    report_progress()
    set_digital_out(0, True)
    new_pose = pose_trans(tuft_coords, p[0.5915, 0.8585, -0.0020, 0, 0, 0])
    movel(p[new_pose[0], new_pose[1], new_pose[2], current_pose[3], current_pose[4], current_pose[5]], a=1.2, v=0.0600)
    report_progress()
    set_digital_out(0, False)
    new_pose = pose_trans(tuft_coords, p[0.5915, 0.8585, 0.1500, 0, 0, 0])
    movel(p[new_pose[0], new_pose[1], new_pose[2], current_pose[3], current_pose[4], current_pose[5]], a=0.8, v=0.2000)
    report_progress()
    new_pose = pose_trans(tuft_coords, p[0.5935, 0.1895, 0.1500, 0, 0, 0])
    movel(p[new_pose[0], new_pose[1], new_pose[2], current_pose[3], current_pose[4], current_pose[5]], a=1.2, v=0.2000)
    report_progress()
    new_pose = pose_trans(tuft_coords, p[0.5935, 0.1895, -0.0020, 0, 0, 0])
    movel(p[new_pose[0], new_pose[1], new_pose[2], current_pose[3], current_pose[4], current_pose[5]], a=0.8, v=0.2000)
    report_progress()
    set_digital_out(0, True)
    new_pose = pose_trans(tuft_coords, p[0.5935, 0.8605, -0.0020, 0, 0, 0])
    movel(p[new_pose[0], new_pose[1], new_pose[2], current_pose[3], current_pose[4], current_pose[5]], a=1.2, v=0.0600)
    report_progress()
    set_digital_out(0, False)
    new_pose = pose_trans(tuft_coords, p[0.5935, 0.8605, 0.1500, 0, 0, 0])
    movel(p[new_pose[0], new_pose[1], new_pose[2], current_pose[3], current_pose[4], current_pose[5]], a=0.8, v=0.2000)
    report_progress()
    new_pose = pose_trans(tuft_coords, p[0.5954, 0.1895, 0.1500, 0, 0, 0])
    movel(p[new_pose[0], new_pose[1], new_pose[2], current_pose[3], current_pose[4], current_pose[5]], a=1.2, v=0.2000)
    report_progress()
    new_pose = pose_trans(tuft_coords, p[0.5954, 0.1895, -0.0020, 0, 0, 0])
    movel(p[new_pose[0], new_pose[1], new_pose[2], current_pose[3], current_pose[4], current_pose[5]], a=0.8, v=0.2000)
    report_progress()
    set_digital_out(0, True)
    new_pose = pose_trans(tuft_coords, p[0.5954, 0.8605, -0.0020, 0, 0, 0])
    movel(p[new_pose[0], new_pose[1], new_pose[2], current_pose[3], current_pose[4], current_pose[5]], a=1.2, v=0.0600)
    report_progress()
    set_digital_out(0, False)
    new_pose = pose_trans(tuft_coords, p[0.5954, 0.8605, 0.1500, 0, 0, 0])
    movel(p[new_pose[0], new_pose[1], new_pose[2], current_pose[3], current_pose[4], current_pose[5]], a=0.8, v=0.2000)
    report_progress()
    new_pose = pose_trans(tuft_coords, p[0.5974, 0.1876, 0.1500, 0, 0, 0])
    movel(p[new_pose[0], new_pose[1], new_pose[2], current_pose[3], current_pose[4], current_pose[5]], a=1.2, v=0.2000)
    report_progress()
    new_pose = pose_trans(tuft_coords, p[0.5974, 0.1876, -0.0020, 0, 0, 0])
    movel(p[new_pose[0], new_pose[1], new_pose[2], current_pose[3], current_pose[4], current_pose[5]], a=0.8, v=0.2000)
    report_progress()
    set_digital_out(0, True)
    new_pose = pose_trans(tuft_coords, p[0.5974, 0.8624, -0.0020, 0, 0, 0])
    movel(p[new_pose[0], new_pose[1], new_pose[2], current_pose[3], current_pose[4], current_pose[5]], a=1.2, v=0.0600)
    report_progress()
    set_digital_out(0, False)
    new_pose = pose_trans(tuft_coords, p[0.5974, 0.8624, 0.1500, 0, 0, 0])
    movel(p[new_pose[0], new_pose[1], new_pose[2], current_pose[3], current_pose[4], current_pose[5]], a=0.8, v=0.2000)
    report_progress()
    new_pose = pose_trans(tuft_coords, p[0.5993, 0.1876, 0.1500, 0, 0, 0])
    movel(p[new_pose[0], new_pose[1], new_pose[2], current_pose[3], current_pose[4], current_pose[5]], a=1.2, v=0.2000)
    report_progress()
    new_pose = pose_trans(tuft_coords, p[0.5993, 0.1876, -0.0020, 0, 0, 0])
    movel(p[new_pose[0], new_pose[1], new_pose[2], current_pose[3], current_pose[4], current_pose[5]], a=0.8, v=0.2000)
    report_progress()
    set_digital_out(0, True)
    new_pose = pose_trans(tuft_coords, p[0.5993, 0.8624, -0.0020, 0, 0, 0])
    movel(p[new_pose[0], new_pose[1], new_pose[2], current_pose[3], current_pose[4], current_pose[5]], a=1.2, v=0.0600)
    report_progress()
    set_digital_out(0, False)
    new_pose = pose_trans(tuft_coords, p[0.5993, 0.8624, 0.1500, 0, 0, 0])
    movel(p[new_pose[0], new_pose[1], new_pose[2], current_pose[3], current_pose[4], current_pose[5]], a=0.8, v=0.2000)
    report_progress()
    new_pose = pose_trans(tuft_coords, p[0.6012, 0.1856, 0.1500, 0, 0, 0])
    movel(p[new_pose[0], new_pose[1], new_pose[2], current_pose[3], current_pose[4], current_pose[5]], a=1.2, v=0.2000)
    report_progress()
    new_pose = pose_trans(tuft_coords, p[0.6012, 0.1856, -0.0020, 0, 0, 0])
    movel(p[new_pose[0], new_pose[1], new_pose[2], current_pose[3], current_pose[4], current_pose[5]], a=0.8, v=0.2000)
    report_progress()
    set_digital_out(0, True)
    new_pose = pose_trans(tuft_coords, p[0.6012, 0.8644, -0.0020, 0, 0, 0])
    movel(p[new_pose[0], new_pose[1], new_pose[2], current_pose[3], current_pose[4], current_pose[5]], a=1.2, v=0.0600)
    report_progress()
    set_digital_out(0, False)
    new_pose = pose_trans(tuft_coords, p[0.6012, 0.8644, 0.1500, 0, 0, 0])
    movel(p[new_pose[0], new_pose[1], new_pose[2], current_pose[3], current_pose[4], current_pose[5]], a=0.8, v=0.2000)
    report_progress()
    new_pose = pose_trans(tuft_coords, p[0.6032, 0.1856, 0.1500, 0, 0, 0])
    movel(p[new_pose[0], new_pose[1], new_pose[2], current_pose[3], current_pose[4], current_pose[5]], a=1.2, v=0.2000)
    report_progress()
    new_pose = pose_trans(tuft_coords, p[0.6032, 0.1856, -0.0020, 0, 0, 0])
    movel(p[new_pose[0], new_pose[1], new_pose[2], current_pose[3], current_pose[4], current_pose[5]], a=0.8, v=0.2000)
    report_progress()
    set_digital_out(0, True)
    new_pose = pose_trans(tuft_coords, p[0.6032, 0.8644, -0.0020, 0, 0, 0])
    movel(p[new_pose[0], new_pose[1], new_pose[2], current_pose[3], current_pose[4], current_pose[5]], a=1.2, v=0.0600)
    report_progress()
    set_digital_out(0, False)
    new_pose = pose_trans(tuft_coords, p[0.6032, 0.8644, 0.1500, 0, 0, 0])
    movel(p[new_pose[0], new_pose[1], new_pose[2], current_pose[3], current_pose[4], current_pose[5]], a=0.8, v=0.2000)
    report_progress()
    new_pose = pose_trans(tuft_coords, p[0.6051, 0.1856, 0.1500, 0, 0, 0])
    movel(p[new_pose[0], new_pose[1], new_pose[2], current_pose[3], current_pose[4], current_pose[5]], a=1.2, v=0.2000)
    report_progress()
    new_pose = pose_trans(tuft_coords, p[0.6051, 0.1856, -0.0020, 0, 0, 0])
    movel(p[new_pose[0], new_pose[1], new_pose[2], current_pose[3], current_pose[4], current_pose[5]], a=0.8, v=0.2000)
    report_progress()
    set_digital_out(0, True)
    new_pose = pose_trans(tuft_coords, p[0.6051, 0.8644, -0.0020, 0, 0, 0])
    movel(p[new_pose[0], new_pose[1], new_pose[2], current_pose[3], current_pose[4], current_pose[5]], a=1.2, v=0.0600)
    report_progress()
    set_digital_out(0, False)
    new_pose = pose_trans(tuft_coords, p[0.6051, 0.8644, 0.1500, 0, 0, 0])
    movel(p[new_pose[0], new_pose[1], new_pose[2], current_pose[3], current_pose[4], current_pose[5]], a=0.8, v=0.2000)
    report_progress()
    new_pose = pose_trans(tuft_coords, p[0.6071, 0.1836, 0.1500, 0, 0, 0])
    movel(p[new_pose[0], new_pose[1], new_pose[2], current_pose[3], current_pose[4], current_pose[5]], a=1.2, v=0.2000)
    report_progress()
    new_pose = pose_trans(tuft_coords, p[0.6071, 0.1836, -0.0020, 0, 0, 0])
    movel(p[new_pose[0], new_pose[1], new_pose[2], current_pose[3], current_pose[4], current_pose[5]], a=0.8, v=0.2000)
    report_progress()
    set_digital_out(0, True)
    new_pose = pose_trans(tuft_coords, p[0.6071, 0.8664, -0.0020, 0, 0, 0])
    movel(p[new_pose[0], new_pose[1], new_pose[2], current_pose[3], current_pose[4], current_pose[5]], a=1.2, v=0.0600)
    report_progress()
    set_digital_out(0, False)
    new_pose = pose_trans(tuft_coords, p[0.6071, 0.8664, 0.1500, 0, 0, 0])
    movel(p[new_pose[0], new_pose[1], new_pose[2], current_pose[3], current_pose[4], current_pose[5]], a=0.8, v=0.2000)
    report_progress()
    new_pose = pose_trans(tuft_coords, p[0.6090, 0.1836, 0.1500, 0, 0, 0])
    movel(p[new_pose[0], new_pose[1], new_pose[2], current_pose[3], current_pose[4], current_pose[5]], a=1.2, v=0.2000)
    report_progress()
    new_pose = pose_trans(tuft_coords, p[0.6090, 0.1836, -0.0020, 0, 0, 0])
    movel(p[new_pose[0], new_pose[1], new_pose[2], current_pose[3], current_pose[4], current_pose[5]], a=0.8, v=0.2000)
    report_progress()
    set_digital_out(0, True)
    new_pose = pose_trans(tuft_coords, p[0.6090, 0.8664, -0.0020, 0, 0, 0])
    movel(p[new_pose[0], new_pose[1], new_pose[2], current_pose[3], current_pose[4], current_pose[5]], a=1.2, v=0.0600)
    report_progress()
    set_digital_out(0, False)
    new_pose = pose_trans(tuft_coords, p[0.6090, 0.8664, 0.1500, 0, 0, 0])
    movel(p[new_pose[0], new_pose[1], new_pose[2], current_pose[3], current_pose[4], current_pose[5]], a=0.8, v=0.2000)
    report_progress()
    new_pose = pose_trans(tuft_coords, p[0.6110, 0.1816, 0.1500, 0, 0, 0])
    movel(p[new_pose[0], new_pose[1], new_pose[2], current_pose[3], current_pose[4], current_pose[5]], a=1.2, v=0.2000)
    report_progress()
    new_pose = pose_trans(tuft_coords, p[0.6110, 0.1816, -0.0020, 0, 0, 0])
    movel(p[new_pose[0], new_pose[1], new_pose[2], current_pose[3], current_pose[4], current_pose[5]], a=0.8, v=0.2000)
    report_progress()
    set_digital_out(0, True)
    new_pose = pose_trans(tuft_coords, p[0.6110, 0.8684, -0.0020, 0, 0, 0])
    movel(p[new_pose[0], new_pose[1], new_pose[2], current_pose[3], current_pose[4], current_pose[5]], a=1.2, v=0.0600)
    report_progress()
    set_digital_out(0, False)
    new_pose = pose_trans(tuft_coords, p[0.6110, 0.8684, 0.1500, 0, 0, 0])
    movel(p[new_pose[0], new_pose[1], new_pose[2], current_pose[3], current_pose[4], current_pose[5]], a=0.8, v=0.2000)
    report_progress()
    new_pose = pose_trans(tuft_coords, p[0.6129, 0.1816, 0.1500, 0, 0, 0])
    movel(p[new_pose[0], new_pose[1], new_pose[2], current_pose[3], current_pose[4], current_pose[5]], a=1.2, v=0.2000)
    report_progress()
    new_pose = pose_trans(tuft_coords, p[0.6129, 0.1816, -0.0020, 0, 0, 0])
    movel(p[new_pose[0], new_pose[1], new_pose[2], current_pose[3], current_pose[4], current_pose[5]], a=0.8, v=0.2000)
    report_progress()
    set_digital_out(0, True)
    new_pose = pose_trans(tuft_coords, p[0.6129, 0.8684, -0.0020, 0, 0, 0])
    movel(p[new_pose[0], new_pose[1], new_pose[2], current_pose[3], current_pose[4], current_pose[5]], a=1.2, v=0.0600)
    report_progress()
    set_digital_out(0, False)
    new_pose = pose_trans(tuft_coords, p[0.6129, 0.8684, 0.1500, 0, 0, 0])
    movel(p[new_pose[0], new_pose[1], new_pose[2], current_pose[3], current_pose[4], current_pose[5]], a=0.8, v=0.2000)
    report_progress()
    new_pose = pose_trans(tuft_coords, p[0.6149, 0.1816, 0.1500, 0, 0, 0])
    movel(p[new_pose[0], new_pose[1], new_pose[2], current_pose[3], current_pose[4], current_pose[5]], a=1.2, v=0.2000)
    report_progress()
    new_pose = pose_trans(tuft_coords, p[0.6149, 0.1816, -0.0020, 0, 0, 0])
    movel(p[new_pose[0], new_pose[1], new_pose[2], current_pose[3], current_pose[4], current_pose[5]], a=0.8, v=0.2000)
    report_progress()
    set_digital_out(0, True)
    new_pose = pose_trans(tuft_coords, p[0.6149, 0.8684, -0.0020, 0, 0, 0])
    movel(p[new_pose[0], new_pose[1], new_pose[2], current_pose[3], current_pose[4], current_pose[5]], a=1.2, v=0.0600)
    report_progress()
    set_digital_out(0, False)
    new_pose = pose_trans(tuft_coords, p[0.6149, 0.8684, 0.1500, 0, 0, 0])
    movel(p[new_pose[0], new_pose[1], new_pose[2], current_pose[3], current_pose[4], current_pose[5]], a=0.8, v=0.2000)
    report_progress()
    new_pose = pose_trans(tuft_coords, p[0.6168, 0.1796, 0.1500, 0, 0, 0])
    movel(p[new_pose[0], new_pose[1], new_pose[2], current_pose[3], current_pose[4], current_pose[5]], a=1.2, v=0.2000)
    report_progress()
    new_pose = pose_trans(tuft_coords, p[0.6168, 0.1796, -0.0020, 0, 0, 0])
    movel(p[new_pose[0], new_pose[1], new_pose[2], current_pose[3], current_pose[4], current_pose[5]], a=0.8, v=0.2000)
    report_progress()
    set_digital_out(0, True)
    new_pose = pose_trans(tuft_coords, p[0.6168, 0.8704, -0.0020, 0, 0, 0])
    movel(p[new_pose[0], new_pose[1], new_pose[2], current_pose[3], current_pose[4], current_pose[5]], a=1.2, v=0.0600)
    report_progress()
    set_digital_out(0, False)
    new_pose = pose_trans(tuft_coords, p[0.6168, 0.8704, 0.1500, 0, 0, 0])
    movel(p[new_pose[0], new_pose[1], new_pose[2], current_pose[3], current_pose[4], current_pose[5]], a=0.8, v=0.2000)
    report_progress()
    new_pose = pose_trans(tuft_coords, p[0.6188, 0.1796, 0.1500, 0, 0, 0])
    movel(p[new_pose[0], new_pose[1], new_pose[2], current_pose[3], current_pose[4], current_pose[5]], a=1.2, v=0.2000)
    report_progress()
    new_pose = pose_trans(tuft_coords, p[0.6188, 0.1796, -0.0020, 0, 0, 0])
    movel(p[new_pose[0], new_pose[1], new_pose[2], current_pose[3], current_pose[4], current_pose[5]], a=0.8, v=0.2000)
    report_progress()
    set_digital_out(0, True)
    new_pose = pose_trans(tuft_coords, p[0.6188, 0.8704, -0.0020, 0, 0, 0])
    movel(p[new_pose[0], new_pose[1], new_pose[2], current_pose[3], current_pose[4], current_pose[5]], a=1.2, v=0.0600)
    report_progress()
    set_digital_out(0, False)
    new_pose = pose_trans(tuft_coords, p[0.6188, 0.8704, 0.1500, 0, 0, 0])
    movel(p[new_pose[0], new_pose[1], new_pose[2], current_pose[3], current_pose[4], current_pose[5]], a=0.8, v=0.2000)
    report_progress()
    new_pose = pose_trans(tuft_coords, p[0.6207, 0.1777, 0.1500, 0, 0, 0])
    movel(p[new_pose[0], new_pose[1], new_pose[2], current_pose[3], current_pose[4], current_pose[5]], a=1.2, v=0.2000)
    report_progress()
    new_pose = pose_trans(tuft_coords, p[0.6207, 0.1777, -0.0020, 0, 0, 0])
    movel(p[new_pose[0], new_pose[1], new_pose[2], current_pose[3], current_pose[4], current_pose[5]], a=0.8, v=0.2000)
    report_progress()
    set_digital_out(0, True)
    new_pose = pose_trans(tuft_coords, p[0.6207, 0.8723, -0.0020, 0, 0, 0])
    movel(p[new_pose[0], new_pose[1], new_pose[2], current_pose[3], current_pose[4], current_pose[5]], a=1.2, v=0.0600)
    report_progress()
    set_digital_out(0, False)
    new_pose = pose_trans(tuft_coords, p[0.6207, 0.8723, 0.1500, 0, 0, 0])
    movel(p[new_pose[0], new_pose[1], new_pose[2], current_pose[3], current_pose[4], current_pose[5]], a=0.8, v=0.2000)
    report_progress()
    new_pose = pose_trans(tuft_coords, p[0.6226, 0.1777, 0.1500, 0, 0, 0])
    movel(p[new_pose[0], new_pose[1], new_pose[2], current_pose[3], current_pose[4], current_pose[5]], a=1.2, v=0.2000)
    report_progress()
    new_pose = pose_trans(tuft_coords, p[0.6226, 0.1777, -0.0020, 0, 0, 0])
    movel(p[new_pose[0], new_pose[1], new_pose[2], current_pose[3], current_pose[4], current_pose[5]], a=0.8, v=0.2000)
    report_progress()
    set_digital_out(0, True)
    new_pose = pose_trans(tuft_coords, p[0.6226, 0.8723, -0.0020, 0, 0, 0])
    movel(p[new_pose[0], new_pose[1], new_pose[2], current_pose[3], current_pose[4], current_pose[5]], a=1.2, v=0.0600)
    report_progress()
    set_digital_out(0, False)
    new_pose = pose_trans(tuft_coords, p[0.6226, 0.8723, 0.1500, 0, 0, 0])
    movel(p[new_pose[0], new_pose[1], new_pose[2], current_pose[3], current_pose[4], current_pose[5]], a=0.8, v=0.2000)
    report_progress()
    new_pose = pose_trans(tuft_coords, p[0.6246, 0.1777, 0.1500, 0, 0, 0])
    movel(p[new_pose[0], new_pose[1], new_pose[2], current_pose[3], current_pose[4], current_pose[5]], a=1.2, v=0.2000)
    report_progress()
    new_pose = pose_trans(tuft_coords, p[0.6246, 0.1777, -0.0020, 0, 0, 0])
    movel(p[new_pose[0], new_pose[1], new_pose[2], current_pose[3], current_pose[4], current_pose[5]], a=0.8, v=0.2000)
    report_progress()
    set_digital_out(0, True)
    new_pose = pose_trans(tuft_coords, p[0.6246, 0.8723, -0.0020, 0, 0, 0])
    movel(p[new_pose[0], new_pose[1], new_pose[2], current_pose[3], current_pose[4], current_pose[5]], a=1.2, v=0.0600)
    report_progress()
    set_digital_out(0, False)
    new_pose = pose_trans(tuft_coords, p[0.6246, 0.8723, 0.1500, 0, 0, 0])
    movel(p[new_pose[0], new_pose[1], new_pose[2], current_pose[3], current_pose[4], current_pose[5]], a=0.8, v=0.2000)
    report_progress()
    new_pose = pose_trans(tuft_coords, p[0.6265, 0.1757, 0.1500, 0, 0, 0])
    movel(p[new_pose[0], new_pose[1], new_pose[2], current_pose[3], current_pose[4], current_pose[5]], a=1.2, v=0.2000)
    report_progress()
    new_pose = pose_trans(tuft_coords, p[0.6265, 0.1757, -0.0020, 0, 0, 0])
    movel(p[new_pose[0], new_pose[1], new_pose[2], current_pose[3], current_pose[4], current_pose[5]], a=0.8, v=0.2000)
    report_progress()
    set_digital_out(0, True)
    new_pose = pose_trans(tuft_coords, p[0.6265, 0.8743, -0.0020, 0, 0, 0])
    movel(p[new_pose[0], new_pose[1], new_pose[2], current_pose[3], current_pose[4], current_pose[5]], a=1.2, v=0.0600)
    report_progress()
    set_digital_out(0, False)
    new_pose = pose_trans(tuft_coords, p[0.6265, 0.8743, 0.1500, 0, 0, 0])
    movel(p[new_pose[0], new_pose[1], new_pose[2], current_pose[3], current_pose[4], current_pose[5]], a=0.8, v=0.2000)
    report_progress()
    new_pose = pose_trans(tuft_coords, p[0.6285, 0.1757, 0.1500, 0, 0, 0])
    movel(p[new_pose[0], new_pose[1], new_pose[2], current_pose[3], current_pose[4], current_pose[5]], a=1.2, v=0.2000)
    report_progress()
    new_pose = pose_trans(tuft_coords, p[0.6285, 0.1757, -0.0020, 0, 0, 0])
    movel(p[new_pose[0], new_pose[1], new_pose[2], current_pose[3], current_pose[4], current_pose[5]], a=0.8, v=0.2000)
    report_progress()
    set_digital_out(0, True)
    new_pose = pose_trans(tuft_coords, p[0.6285, 0.8743, -0.0020, 0, 0, 0])
    movel(p[new_pose[0], new_pose[1], new_pose[2], current_pose[3], current_pose[4], current_pose[5]], a=1.2, v=0.0600)
    report_progress()
    set_digital_out(0, False)
    new_pose = pose_trans(tuft_coords, p[0.6285, 0.8743, 0.1500, 0, 0, 0])
    movel(p[new_pose[0], new_pose[1], new_pose[2], current_pose[3], current_pose[4], current_pose[5]], a=0.8, v=0.2000)
    report_progress()
    new_pose = pose_trans(tuft_coords, p[0.6304, 0.1757, 0.1500, 0, 0, 0])
    movel(p[new_pose[0], new_pose[1], new_pose[2], current_pose[3], current_pose[4], current_pose[5]], a=1.2, v=0.2000)
    report_progress()
    new_pose = pose_trans(tuft_coords, p[0.6304, 0.1757, -0.0020, 0, 0, 0])
    movel(p[new_pose[0], new_pose[1], new_pose[2], current_pose[3], current_pose[4], current_pose[5]], a=0.8, v=0.2000)
    report_progress()
    set_digital_out(0, True)
    new_pose = pose_trans(tuft_coords, p[0.6304, 0.8743, -0.0020, 0, 0, 0])
    movel(p[new_pose[0], new_pose[1], new_pose[2], current_pose[3], current_pose[4], current_pose[5]], a=1.2, v=0.0600)
    report_progress()
    set_digital_out(0, False)
    new_pose = pose_trans(tuft_coords, p[0.6304, 0.8743, 0.1500, 0, 0, 0])
    movel(p[new_pose[0], new_pose[1], new_pose[2], current_pose[3], current_pose[4], current_pose[5]], a=0.8, v=0.2000)
    report_progress()
    new_pose = pose_trans(tuft_coords, p[0.6324, 0.1737, 0.1500, 0, 0, 0])
    movel(p[new_pose[0], new_pose[1], new_pose[2], current_pose[3], current_pose[4], current_pose[5]], a=1.2, v=0.2000)
    report_progress()
    new_pose = pose_trans(tuft_coords, p[0.6324, 0.1737, -0.0020, 0, 0, 0])
    movel(p[new_pose[0], new_pose[1], new_pose[2], current_pose[3], current_pose[4], current_pose[5]], a=0.8, v=0.2000)
    report_progress()
    set_digital_out(0, True)
    new_pose = pose_trans(tuft_coords, p[0.6324, 0.8763, -0.0020, 0, 0, 0])
    movel(p[new_pose[0], new_pose[1], new_pose[2], current_pose[3], current_pose[4], current_pose[5]], a=1.2, v=0.0600)
    report_progress()
    set_digital_out(0, False)
    new_pose = pose_trans(tuft_coords, p[0.6324, 0.8763, 0.1500, 0, 0, 0])
    movel(p[new_pose[0], new_pose[1], new_pose[2], current_pose[3], current_pose[4], current_pose[5]], a=0.8, v=0.2000)
    report_progress()
    new_pose = pose_trans(tuft_coords, p[0.6343, 0.1737, 0.1500, 0, 0, 0])
    movel(p[new_pose[0], new_pose[1], new_pose[2], current_pose[3], current_pose[4], current_pose[5]], a=1.2, v=0.2000)
    report_progress()
    new_pose = pose_trans(tuft_coords, p[0.6343, 0.1737, -0.0020, 0, 0, 0])
    movel(p[new_pose[0], new_pose[1], new_pose[2], current_pose[3], current_pose[4], current_pose[5]], a=0.8, v=0.2000)
    report_progress()
    set_digital_out(0, True)
    new_pose = pose_trans(tuft_coords, p[0.6343, 0.8763, -0.0020, 0, 0, 0])
    movel(p[new_pose[0], new_pose[1], new_pose[2], current_pose[3], current_pose[4], current_pose[5]], a=1.2, v=0.0600)
    report_progress()
    set_digital_out(0, False)
    new_pose = pose_trans(tuft_coords, p[0.6343, 0.8763, 0.1500, 0, 0, 0])
    movel(p[new_pose[0], new_pose[1], new_pose[2], current_pose[3], current_pose[4], current_pose[5]], a=0.8, v=0.2000)
    report_progress()
    new_pose = pose_trans(tuft_coords, p[0.6362, 0.1737, 0.1500, 0, 0, 0])
    movel(p[new_pose[0], new_pose[1], new_pose[2], current_pose[3], current_pose[4], current_pose[5]], a=1.2, v=0.2000)
    report_progress()
    new_pose = pose_trans(tuft_coords, p[0.6362, 0.1737, -0.0020, 0, 0, 0])
    movel(p[new_pose[0], new_pose[1], new_pose[2], current_pose[3], current_pose[4], current_pose[5]], a=0.8, v=0.2000)
    report_progress()
    set_digital_out(0, True)
    new_pose = pose_trans(tuft_coords, p[0.6362, 0.8763, -0.0020, 0, 0, 0])
    movel(p[new_pose[0], new_pose[1], new_pose[2], current_pose[3], current_pose[4], current_pose[5]], a=1.2, v=0.0600)
    report_progress()
    set_digital_out(0, False)
    new_pose = pose_trans(tuft_coords, p[0.6362, 0.8763, 0.1500, 0, 0, 0])
    movel(p[new_pose[0], new_pose[1], new_pose[2], current_pose[3], current_pose[4], current_pose[5]], a=0.8, v=0.2000)
    report_progress()
    new_pose = pose_trans(tuft_coords, p[0.6382, 0.1717, 0.1500, 0, 0, 0])
    movel(p[new_pose[0], new_pose[1], new_pose[2], current_pose[3], current_pose[4], current_pose[5]], a=1.2, v=0.2000)
    report_progress()
    new_pose = pose_trans(tuft_coords, p[0.6382, 0.1717, -0.0020, 0, 0, 0])
    movel(p[new_pose[0], new_pose[1], new_pose[2], current_pose[3], current_pose[4], current_pose[5]], a=0.8, v=0.2000)
    report_progress()
    set_digital_out(0, True)
    new_pose = pose_trans(tuft_coords, p[0.6382, 0.8783, -0.0020, 0, 0, 0])
    movel(p[new_pose[0], new_pose[1], new_pose[2], current_pose[3], current_pose[4], current_pose[5]], a=1.2, v=0.0600)
    report_progress()
    set_digital_out(0, False)
    new_pose = pose_trans(tuft_coords, p[0.6382, 0.8783, 0.1500, 0, 0, 0])
    movel(p[new_pose[0], new_pose[1], new_pose[2], current_pose[3], current_pose[4], current_pose[5]], a=0.8, v=0.2000)
    report_progress()
    new_pose = pose_trans(tuft_coords, p[0.6401, 0.1717, 0.1500, 0, 0, 0])
    movel(p[new_pose[0], new_pose[1], new_pose[2], current_pose[3], current_pose[4], current_pose[5]], a=1.2, v=0.2000)
    report_progress()
    new_pose = pose_trans(tuft_coords, p[0.6401, 0.1717, -0.0020, 0, 0, 0])
    movel(p[new_pose[0], new_pose[1], new_pose[2], current_pose[3], current_pose[4], current_pose[5]], a=0.8, v=0.2000)
    report_progress()
    set_digital_out(0, True)
    new_pose = pose_trans(tuft_coords, p[0.6401, 0.8783, -0.0020, 0, 0, 0])
    movel(p[new_pose[0], new_pose[1], new_pose[2], current_pose[3], current_pose[4], current_pose[5]], a=1.2, v=0.0600)
    report_progress()
    set_digital_out(0, False)
    new_pose = pose_trans(tuft_coords, p[0.6401, 0.8783, 0.1500, 0, 0, 0])
    movel(p[new_pose[0], new_pose[1], new_pose[2], current_pose[3], current_pose[4], current_pose[5]], a=0.8, v=0.2000)
    report_progress()
    new_pose = pose_trans(tuft_coords, p[0.6421, 0.1717, 0.1500, 0, 0, 0])
    movel(p[new_pose[0], new_pose[1], new_pose[2], current_pose[3], current_pose[4], current_pose[5]], a=1.2, v=0.2000)
    report_progress()
    new_pose = pose_trans(tuft_coords, p[0.6421, 0.1717, -0.0020, 0, 0, 0])
    movel(p[new_pose[0], new_pose[1], new_pose[2], current_pose[3], current_pose[4], current_pose[5]], a=0.8, v=0.2000)
    report_progress()
    set_digital_out(0, True)
    new_pose = pose_trans(tuft_coords, p[0.6421, 0.8783, -0.0020, 0, 0, 0])
    movel(p[new_pose[0], new_pose[1], new_pose[2], current_pose[3], current_pose[4], current_pose[5]], a=1.2, v=0.0600)
    report_progress()
    set_digital_out(0, False)
    new_pose = pose_trans(tuft_coords, p[0.6421, 0.8783, 0.1500, 0, 0, 0])
    movel(p[new_pose[0], new_pose[1], new_pose[2], current_pose[3], current_pose[4], current_pose[5]], a=0.8, v=0.2000)
    report_progress()
    new_pose = pose_trans(tuft_coords, p[0.6440, 0.1697, 0.1500, 0, 0, 0])
    movel(p[new_pose[0], new_pose[1], new_pose[2], current_pose[3], current_pose[4], current_pose[5]], a=1.2, v=0.2000)
    report_progress()
    new_pose = pose_trans(tuft_coords, p[0.6440, 0.1697, -0.0020, 0, 0, 0])
    movel(p[new_pose[0], new_pose[1], new_pose[2], current_pose[3], current_pose[4], current_pose[5]], a=0.8, v=0.2000)
    report_progress()
    set_digital_out(0, True)
    new_pose = pose_trans(tuft_coords, p[0.6440, 0.8803, -0.0020, 0, 0, 0])
    movel(p[new_pose[0], new_pose[1], new_pose[2], current_pose[3], current_pose[4], current_pose[5]], a=1.2, v=0.0600)
    report_progress()
    set_digital_out(0, False)
    new_pose = pose_trans(tuft_coords, p[0.6440, 0.8803, 0.1500, 0, 0, 0])
    movel(p[new_pose[0], new_pose[1], new_pose[2], current_pose[3], current_pose[4], current_pose[5]], a=0.8, v=0.2000)
    report_progress()
    new_pose = pose_trans(tuft_coords, p[0.6460, 0.1697, 0.1500, 0, 0, 0])
    movel(p[new_pose[0], new_pose[1], new_pose[2], current_pose[3], current_pose[4], current_pose[5]], a=1.2, v=0.2000)
    report_progress()
    new_pose = pose_trans(tuft_coords, p[0.6460, 0.1697, -0.0020, 0, 0, 0])
    movel(p[new_pose[0], new_pose[1], new_pose[2], current_pose[3], current_pose[4], current_pose[5]], a=0.8, v=0.2000)
    report_progress()
    set_digital_out(0, True)
    new_pose = pose_trans(tuft_coords, p[0.6460, 0.8803, -0.0020, 0, 0, 0])
    movel(p[new_pose[0], new_pose[1], new_pose[2], current_pose[3], current_pose[4], current_pose[5]], a=1.2, v=0.0600)
    report_progress()
    set_digital_out(0, False)
    new_pose = pose_trans(tuft_coords, p[0.6460, 0.8803, 0.1500, 0, 0, 0])
    movel(p[new_pose[0], new_pose[1], new_pose[2], current_pose[3], current_pose[4], current_pose[5]], a=0.8, v=0.2000)
    report_progress()
    new_pose = pose_trans(tuft_coords, p[0.6479, 0.1697, 0.1500, 0, 0, 0])
    movel(p[new_pose[0], new_pose[1], new_pose[2], current_pose[3], current_pose[4], current_pose[5]], a=1.2, v=0.2000)
    report_progress()
    new_pose = pose_trans(tuft_coords, p[0.6479, 0.1697, -0.0020, 0, 0, 0])
    movel(p[new_pose[0], new_pose[1], new_pose[2], current_pose[3], current_pose[4], current_pose[5]], a=0.8, v=0.2000)
    report_progress()
    set_digital_out(0, True)
    new_pose = pose_trans(tuft_coords, p[0.6479, 0.8803, -0.0020, 0, 0, 0])
    movel(p[new_pose[0], new_pose[1], new_pose[2], current_pose[3], current_pose[4], current_pose[5]], a=1.2, v=0.0600)
    report_progress()
    set_digital_out(0, False)
    new_pose = pose_trans(tuft_coords, p[0.6479, 0.8803, 0.1500, 0, 0, 0])
    movel(p[new_pose[0], new_pose[1], new_pose[2], current_pose[3], current_pose[4], current_pose[5]], a=0.8, v=0.2000)
    report_progress()
    new_pose = pose_trans(tuft_coords, p[0.6499, 0.1678, 0.1500, 0, 0, 0])
    movel(p[new_pose[0], new_pose[1], new_pose[2], current_pose[3], current_pose[4], current_pose[5]], a=1.2, v=0.2000)
    report_progress()
    new_pose = pose_trans(tuft_coords, p[0.6499, 0.1678, -0.0020, 0, 0, 0])
    movel(p[new_pose[0], new_pose[1], new_pose[2], current_pose[3], current_pose[4], current_pose[5]], a=0.8, v=0.2000)
    report_progress()
    set_digital_out(0, True)
    new_pose = pose_trans(tuft_coords, p[0.6499, 0.8822, -0.0020, 0, 0, 0])
    movel(p[new_pose[0], new_pose[1], new_pose[2], current_pose[3], current_pose[4], current_pose[5]], a=1.2, v=0.0600)
    report_progress()
    set_digital_out(0, False)
    new_pose = pose_trans(tuft_coords, p[0.6499, 0.8822, 0.1500, 0, 0, 0])
    movel(p[new_pose[0], new_pose[1], new_pose[2], current_pose[3], current_pose[4], current_pose[5]], a=0.8, v=0.2000)
    report_progress()
    new_pose = pose_trans(tuft_coords, p[0.6518, 0.1678, 0.1500, 0, 0, 0])
    movel(p[new_pose[0], new_pose[1], new_pose[2], current_pose[3], current_pose[4], current_pose[5]], a=1.2, v=0.2000)
    report_progress()
    new_pose = pose_trans(tuft_coords, p[0.6518, 0.1678, -0.0020, 0, 0, 0])
    movel(p[new_pose[0], new_pose[1], new_pose[2], current_pose[3], current_pose[4], current_pose[5]], a=0.8, v=0.2000)
    report_progress()
    set_digital_out(0, True)
    new_pose = pose_trans(tuft_coords, p[0.6518, 0.8822, -0.0020, 0, 0, 0])
    movel(p[new_pose[0], new_pose[1], new_pose[2], current_pose[3], current_pose[4], current_pose[5]], a=1.2, v=0.0600)
    report_progress()
    set_digital_out(0, False)
    new_pose = pose_trans(tuft_coords, p[0.6518, 0.8822, 0.1500, 0, 0, 0])
    movel(p[new_pose[0], new_pose[1], new_pose[2], current_pose[3], current_pose[4], current_pose[5]], a=0.8, v=0.2000)
    report_progress()
    new_pose = pose_trans(tuft_coords, p[0.6538, 0.1678, 0.1500, 0, 0, 0])
    movel(p[new_pose[0], new_pose[1], new_pose[2], current_pose[3], current_pose[4], current_pose[5]], a=1.2, v=0.2000)
    report_progress()
    new_pose = pose_trans(tuft_coords, p[0.6538, 0.1678, -0.0020, 0, 0, 0])
    movel(p[new_pose[0], new_pose[1], new_pose[2], current_pose[3], current_pose[4], current_pose[5]], a=0.8, v=0.2000)
    report_progress()
    set_digital_out(0, True)
    new_pose = pose_trans(tuft_coords, p[0.6538, 0.8822, -0.0020, 0, 0, 0])
    movel(p[new_pose[0], new_pose[1], new_pose[2], current_pose[3], current_pose[4], current_pose[5]], a=1.2, v=0.0600)
    report_progress()
    set_digital_out(0, False)
    new_pose = pose_trans(tuft_coords, p[0.6538, 0.8822, 0.1500, 0, 0, 0])
    movel(p[new_pose[0], new_pose[1], new_pose[2], current_pose[3], current_pose[4], current_pose[5]], a=0.8, v=0.2000)
    report_progress()
    new_pose = pose_trans(tuft_coords, p[0.6557, 0.1678, 0.1500, 0, 0, 0])
    movel(p[new_pose[0], new_pose[1], new_pose[2], current_pose[3], current_pose[4], current_pose[5]], a=1.2, v=0.2000)
    report_progress()
    new_pose = pose_trans(tuft_coords, p[0.6557, 0.1678, -0.0020, 0, 0, 0])
    movel(p[new_pose[0], new_pose[1], new_pose[2], current_pose[3], current_pose[4], current_pose[5]], a=0.8, v=0.2000)
    report_progress()
    set_digital_out(0, True)
    new_pose = pose_trans(tuft_coords, p[0.6557, 0.8822, -0.0020, 0, 0, 0])
    movel(p[new_pose[0], new_pose[1], new_pose[2], current_pose[3], current_pose[4], current_pose[5]], a=1.2, v=0.0600)
    report_progress()
    set_digital_out(0, False)
    new_pose = pose_trans(tuft_coords, p[0.6557, 0.8822, 0.1500, 0, 0, 0])
    movel(p[new_pose[0], new_pose[1], new_pose[2], current_pose[3], current_pose[4], current_pose[5]], a=0.8, v=0.2000)
    report_progress()
    new_pose = pose_trans(tuft_coords, p[0.6576, 0.1658, 0.1500, 0, 0, 0])
    movel(p[new_pose[0], new_pose[1], new_pose[2], current_pose[3], current_pose[4], current_pose[5]], a=1.2, v=0.2000)
    report_progress()
    new_pose = pose_trans(tuft_coords, p[0.6576, 0.1658, -0.0020, 0, 0, 0])
    movel(p[new_pose[0], new_pose[1], new_pose[2], current_pose[3], current_pose[4], current_pose[5]], a=0.8, v=0.2000)
    report_progress()
    set_digital_out(0, True)
    new_pose = pose_trans(tuft_coords, p[0.6576, 0.8842, -0.0020, 0, 0, 0])
    movel(p[new_pose[0], new_pose[1], new_pose[2], current_pose[3], current_pose[4], current_pose[5]], a=1.2, v=0.0600)
    report_progress()
    set_digital_out(0, False)
    new_pose = pose_trans(tuft_coords, p[0.6576, 0.8842, 0.1500, 0, 0, 0])
    movel(p[new_pose[0], new_pose[1], new_pose[2], current_pose[3], current_pose[4], current_pose[5]], a=0.8, v=0.2000)
    report_progress()
    new_pose = pose_trans(tuft_coords, p[0.6596, 0.1658, 0.1500, 0, 0, 0])
    movel(p[new_pose[0], new_pose[1], new_pose[2], current_pose[3], current_pose[4], current_pose[5]], a=1.2, v=0.2000)
    report_progress()
    new_pose = pose_trans(tuft_coords, p[0.6596, 0.1658, -0.0020, 0, 0, 0])
    movel(p[new_pose[0], new_pose[1], new_pose[2], current_pose[3], current_pose[4], current_pose[5]], a=0.8, v=0.2000)
    report_progress()
    set_digital_out(0, True)
    new_pose = pose_trans(tuft_coords, p[0.6596, 0.8842, -0.0020, 0, 0, 0])
    movel(p[new_pose[0], new_pose[1], new_pose[2], current_pose[3], current_pose[4], current_pose[5]], a=1.2, v=0.0600)
    report_progress()
    set_digital_out(0, False)
    new_pose = pose_trans(tuft_coords, p[0.6596, 0.8842, 0.1500, 0, 0, 0])
    movel(p[new_pose[0], new_pose[1], new_pose[2], current_pose[3], current_pose[4], current_pose[5]], a=0.8, v=0.2000)
    report_progress()
    new_pose = pose_trans(tuft_coords, p[0.6615, 0.1658, 0.1500, 0, 0, 0])
    movel(p[new_pose[0], new_pose[1], new_pose[2], current_pose[3], current_pose[4], current_pose[5]], a=1.2, v=0.2000)
    report_progress()
    new_pose = pose_trans(tuft_coords, p[0.6615, 0.1658, -0.0020, 0, 0, 0])
    movel(p[new_pose[0], new_pose[1], new_pose[2], current_pose[3], current_pose[4], current_pose[5]], a=0.8, v=0.2000)
    report_progress()
    set_digital_out(0, True)
    new_pose = pose_trans(tuft_coords, p[0.6615, 0.8842, -0.0020, 0, 0, 0])
    movel(p[new_pose[0], new_pose[1], new_pose[2], current_pose[3], current_pose[4], current_pose[5]], a=1.2, v=0.0600)
    report_progress()
    set_digital_out(0, False)
    new_pose = pose_trans(tuft_coords, p[0.6615, 0.8842, 0.1500, 0, 0, 0])
    movel(p[new_pose[0], new_pose[1], new_pose[2], current_pose[3], current_pose[4], current_pose[5]], a=0.8, v=0.2000)
    report_progress()
    new_pose = pose_trans(tuft_coords, p[0.6635, 0.1658, 0.1500, 0, 0, 0])
    movel(p[new_pose[0], new_pose[1], new_pose[2], current_pose[3], current_pose[4], current_pose[5]], a=1.2, v=0.2000)
    report_progress()
    new_pose = pose_trans(tuft_coords, p[0.6635, 0.1658, -0.0020, 0, 0, 0])
    movel(p[new_pose[0], new_pose[1], new_pose[2], current_pose[3], current_pose[4], current_pose[5]], a=0.8, v=0.2000)
    report_progress()
    set_digital_out(0, True)
    new_pose = pose_trans(tuft_coords, p[0.6635, 0.8842, -0.0020, 0, 0, 0])
    movel(p[new_pose[0], new_pose[1], new_pose[2], current_pose[3], current_pose[4], current_pose[5]], a=1.2, v=0.0600)
    report_progress()
    set_digital_out(0, False)
    new_pose = pose_trans(tuft_coords, p[0.6635, 0.8842, 0.1500, 0, 0, 0])
    movel(p[new_pose[0], new_pose[1], new_pose[2], current_pose[3], current_pose[4], current_pose[5]], a=0.8, v=0.2000)
    report_progress()
    new_pose = pose_trans(tuft_coords, p[0.6654, 0.1638, 0.1500, 0, 0, 0])
    movel(p[new_pose[0], new_pose[1], new_pose[2], current_pose[3], current_pose[4], current_pose[5]], a=1.2, v=0.2000)
    report_progress()
    new_pose = pose_trans(tuft_coords, p[0.6654, 0.1638, -0.0020, 0, 0, 0])
    movel(p[new_pose[0], new_pose[1], new_pose[2], current_pose[3], current_pose[4], current_pose[5]], a=0.8, v=0.2000)
    report_progress()
    set_digital_out(0, True)
    new_pose = pose_trans(tuft_coords, p[0.6654, 0.8862, -0.0020, 0, 0, 0])
    movel(p[new_pose[0], new_pose[1], new_pose[2], current_pose[3], current_pose[4], current_pose[5]], a=1.2, v=0.0600)
    report_progress()
    set_digital_out(0, False)
    new_pose = pose_trans(tuft_coords, p[0.6654, 0.8862, 0.1500, 0, 0, 0])
    movel(p[new_pose[0], new_pose[1], new_pose[2], current_pose[3], current_pose[4], current_pose[5]], a=0.8, v=0.2000)
    report_progress()
    new_pose = pose_trans(tuft_coords, p[0.6674, 0.1638, 0.1500, 0, 0, 0])
    movel(p[new_pose[0], new_pose[1], new_pose[2], current_pose[3], current_pose[4], current_pose[5]], a=1.2, v=0.2000)
    report_progress()
    new_pose = pose_trans(tuft_coords, p[0.6674, 0.1638, -0.0020, 0, 0, 0])
    movel(p[new_pose[0], new_pose[1], new_pose[2], current_pose[3], current_pose[4], current_pose[5]], a=0.8, v=0.2000)
    report_progress()
    set_digital_out(0, True)
    new_pose = pose_trans(tuft_coords, p[0.6674, 0.8862, -0.0020, 0, 0, 0])
    movel(p[new_pose[0], new_pose[1], new_pose[2], current_pose[3], current_pose[4], current_pose[5]], a=1.2, v=0.0600)
    report_progress()
    set_digital_out(0, False)
    new_pose = pose_trans(tuft_coords, p[0.6674, 0.8862, 0.1500, 0, 0, 0])
    movel(p[new_pose[0], new_pose[1], new_pose[2], current_pose[3], current_pose[4], current_pose[5]], a=0.8, v=0.2000)
    report_progress()
    new_pose = pose_trans(tuft_coords, p[0.6693, 0.1638, 0.1500, 0, 0, 0])
    movel(p[new_pose[0], new_pose[1], new_pose[2], current_pose[3], current_pose[4], current_pose[5]], a=1.2, v=0.2000)
    report_progress()
    new_pose = pose_trans(tuft_coords, p[0.6693, 0.1638, -0.0020, 0, 0, 0])
    movel(p[new_pose[0], new_pose[1], new_pose[2], current_pose[3], current_pose[4], current_pose[5]], a=0.8, v=0.2000)
    report_progress()
    set_digital_out(0, True)
    new_pose = pose_trans(tuft_coords, p[0.6693, 0.8862, -0.0020, 0, 0, 0])
    movel(p[new_pose[0], new_pose[1], new_pose[2], current_pose[3], current_pose[4], current_pose[5]], a=1.2, v=0.0600)
    report_progress()
    set_digital_out(0, False)
    new_pose = pose_trans(tuft_coords, p[0.6693, 0.8862, 0.1500, 0, 0, 0])
    movel(p[new_pose[0], new_pose[1], new_pose[2], current_pose[3], current_pose[4], current_pose[5]], a=0.8, v=0.2000)
    report_progress()
    new_pose = pose_trans(tuft_coords, p[0.6713, 0.1638, 0.1500, 0, 0, 0])
    movel(p[new_pose[0], new_pose[1], new_pose[2], current_pose[3], current_pose[4], current_pose[5]], a=1.2, v=0.2000)
    report_progress()
    new_pose = pose_trans(tuft_coords, p[0.6713, 0.1638, -0.0020, 0, 0, 0])
    movel(p[new_pose[0], new_pose[1], new_pose[2], current_pose[3], current_pose[4], current_pose[5]], a=0.8, v=0.2000)
    report_progress()
    set_digital_out(0, True)
    new_pose = pose_trans(tuft_coords, p[0.6713, 0.8862, -0.0020, 0, 0, 0])
    movel(p[new_pose[0], new_pose[1], new_pose[2], current_pose[3], current_pose[4], current_pose[5]], a=1.2, v=0.0600)
    report_progress()
    set_digital_out(0, False)
    new_pose = pose_trans(tuft_coords, p[0.6713, 0.8862, 0.1500, 0, 0, 0])
    movel(p[new_pose[0], new_pose[1], new_pose[2], current_pose[3], current_pose[4], current_pose[5]], a=0.8, v=0.2000)
    report_progress()
    new_pose = pose_trans(tuft_coords, p[0.6732, 0.1618, 0.1500, 0, 0, 0])
    movel(p[new_pose[0], new_pose[1], new_pose[2], current_pose[3], current_pose[4], current_pose[5]], a=1.2, v=0.2000)
    report_progress()
    new_pose = pose_trans(tuft_coords, p[0.6732, 0.1618, -0.0020, 0, 0, 0])
    movel(p[new_pose[0], new_pose[1], new_pose[2], current_pose[3], current_pose[4], current_pose[5]], a=0.8, v=0.2000)
    report_progress()
    set_digital_out(0, True)
    new_pose = pose_trans(tuft_coords, p[0.6732, 0.8882, -0.0020, 0, 0, 0])
    movel(p[new_pose[0], new_pose[1], new_pose[2], current_pose[3], current_pose[4], current_pose[5]], a=1.2, v=0.0600)
    report_progress()
    set_digital_out(0, False)
    new_pose = pose_trans(tuft_coords, p[0.6732, 0.8882, 0.1500, 0, 0, 0])
    movel(p[new_pose[0], new_pose[1], new_pose[2], current_pose[3], current_pose[4], current_pose[5]], a=0.8, v=0.2000)
    report_progress()
    new_pose = pose_trans(tuft_coords, p[0.6751, 0.1618, 0.1500, 0, 0, 0])
    movel(p[new_pose[0], new_pose[1], new_pose[2], current_pose[3], current_pose[4], current_pose[5]], a=1.2, v=0.2000)
    report_progress()
    new_pose = pose_trans(tuft_coords, p[0.6751, 0.1618, -0.0020, 0, 0, 0])
    movel(p[new_pose[0], new_pose[1], new_pose[2], current_pose[3], current_pose[4], current_pose[5]], a=0.8, v=0.2000)
    report_progress()
    set_digital_out(0, True)
    new_pose = pose_trans(tuft_coords, p[0.6751, 0.8882, -0.0020, 0, 0, 0])
    movel(p[new_pose[0], new_pose[1], new_pose[2], current_pose[3], current_pose[4], current_pose[5]], a=1.2, v=0.0600)
    report_progress()
    set_digital_out(0, False)
    new_pose = pose_trans(tuft_coords, p[0.6751, 0.8882, 0.1500, 0, 0, 0])
    movel(p[new_pose[0], new_pose[1], new_pose[2], current_pose[3], current_pose[4], current_pose[5]], a=0.8, v=0.2000)
    report_progress()
    new_pose = pose_trans(tuft_coords, p[0.6771, 0.1618, 0.1500, 0, 0, 0])
    movel(p[new_pose[0], new_pose[1], new_pose[2], current_pose[3], current_pose[4], current_pose[5]], a=1.2, v=0.2000)
    report_progress()
    new_pose = pose_trans(tuft_coords, p[0.6771, 0.1618, -0.0020, 0, 0, 0])
    movel(p[new_pose[0], new_pose[1], new_pose[2], current_pose[3], current_pose[4], current_pose[5]], a=0.8, v=0.2000)
    report_progress()
    set_digital_out(0, True)
    new_pose = pose_trans(tuft_coords, p[0.6771, 0.8882, -0.0020, 0, 0, 0])
    movel(p[new_pose[0], new_pose[1], new_pose[2], current_pose[3], current_pose[4], current_pose[5]], a=1.2, v=0.0600)
    report_progress()
    set_digital_out(0, False)
    new_pose = pose_trans(tuft_coords, p[0.6771, 0.8882, 0.1500, 0, 0, 0])
    movel(p[new_pose[0], new_pose[1], new_pose[2], current_pose[3], current_pose[4], current_pose[5]], a=0.8, v=0.2000)
    report_progress()
    new_pose = pose_trans(tuft_coords, p[0.6790, 0.1618, 0.1500, 0, 0, 0])
    movel(p[new_pose[0], new_pose[1], new_pose[2], current_pose[3], current_pose[4], current_pose[5]], a=1.2, v=0.2000)
    report_progress()
    new_pose = pose_trans(tuft_coords, p[0.6790, 0.1618, -0.0020, 0, 0, 0])
    movel(p[new_pose[0], new_pose[1], new_pose[2], current_pose[3], current_pose[4], current_pose[5]], a=0.8, v=0.2000)
    report_progress()
    set_digital_out(0, True)
    new_pose = pose_trans(tuft_coords, p[0.6790, 0.8882, -0.0020, 0, 0, 0])
    movel(p[new_pose[0], new_pose[1], new_pose[2], current_pose[3], current_pose[4], current_pose[5]], a=1.2, v=0.0600)
    report_progress()
    set_digital_out(0, False)
    new_pose = pose_trans(tuft_coords, p[0.6790, 0.8882, 0.1500, 0, 0, 0])
    movel(p[new_pose[0], new_pose[1], new_pose[2], current_pose[3], current_pose[4], current_pose[5]], a=0.8, v=0.2000)
    report_progress()
    new_pose = pose_trans(tuft_coords, p[0.6810, 0.1618, 0.1500, 0, 0, 0])
    movel(p[new_pose[0], new_pose[1], new_pose[2], current_pose[3], current_pose[4], current_pose[5]], a=1.2, v=0.2000)
    report_progress()
    new_pose = pose_trans(tuft_coords, p[0.6810, 0.1618, -0.0020, 0, 0, 0])
    movel(p[new_pose[0], new_pose[1], new_pose[2], current_pose[3], current_pose[4], current_pose[5]], a=0.8, v=0.2000)
    report_progress()
    set_digital_out(0, True)
    new_pose = pose_trans(tuft_coords, p[0.6810, 0.8882, -0.0020, 0, 0, 0])
    movel(p[new_pose[0], new_pose[1], new_pose[2], current_pose[3], current_pose[4], current_pose[5]], a=1.2, v=0.0600)
    report_progress()
    set_digital_out(0, False)
    new_pose = pose_trans(tuft_coords, p[0.6810, 0.8882, 0.1500, 0, 0, 0])
    movel(p[new_pose[0], new_pose[1], new_pose[2], current_pose[3], current_pose[4], current_pose[5]], a=0.8, v=0.2000)
    report_progress()
    new_pose = pose_trans(tuft_coords, p[0.6829, 0.1598, 0.1500, 0, 0, 0])
    movel(p[new_pose[0], new_pose[1], new_pose[2], current_pose[3], current_pose[4], current_pose[5]], a=1.2, v=0.2000)
    report_progress()
    new_pose = pose_trans(tuft_coords, p[0.6829, 0.1598, -0.0020, 0, 0, 0])
    movel(p[new_pose[0], new_pose[1], new_pose[2], current_pose[3], current_pose[4], current_pose[5]], a=0.8, v=0.2000)
    report_progress()
    set_digital_out(0, True)
    new_pose = pose_trans(tuft_coords, p[0.6829, 0.8902, -0.0020, 0, 0, 0])
    movel(p[new_pose[0], new_pose[1], new_pose[2], current_pose[3], current_pose[4], current_pose[5]], a=1.2, v=0.0600)
    report_progress()
    set_digital_out(0, False)
    new_pose = pose_trans(tuft_coords, p[0.6829, 0.8902, 0.1500, 0, 0, 0])
    movel(p[new_pose[0], new_pose[1], new_pose[2], current_pose[3], current_pose[4], current_pose[5]], a=0.8, v=0.2000)
    report_progress()
    new_pose = pose_trans(tuft_coords, p[0.6849, 0.1598, 0.1500, 0, 0, 0])
    movel(p[new_pose[0], new_pose[1], new_pose[2], current_pose[3], current_pose[4], current_pose[5]], a=1.2, v=0.2000)
    report_progress()
    new_pose = pose_trans(tuft_coords, p[0.6849, 0.1598, -0.0020, 0, 0, 0])
    movel(p[new_pose[0], new_pose[1], new_pose[2], current_pose[3], current_pose[4], current_pose[5]], a=0.8, v=0.2000)
    report_progress()
    set_digital_out(0, True)
    new_pose = pose_trans(tuft_coords, p[0.6849, 0.8902, -0.0020, 0, 0, 0])
    movel(p[new_pose[0], new_pose[1], new_pose[2], current_pose[3], current_pose[4], current_pose[5]], a=1.2, v=0.0600)
    report_progress()
    set_digital_out(0, False)
    new_pose = pose_trans(tuft_coords, p[0.6849, 0.8902, 0.1500, 0, 0, 0])
    movel(p[new_pose[0], new_pose[1], new_pose[2], current_pose[3], current_pose[4], current_pose[5]], a=0.8, v=0.2000)
    report_progress()
    new_pose = pose_trans(tuft_coords, p[0.6868, 0.1598, 0.1500, 0, 0, 0])
    movel(p[new_pose[0], new_pose[1], new_pose[2], current_pose[3], current_pose[4], current_pose[5]], a=1.2, v=0.2000)
    report_progress()
    new_pose = pose_trans(tuft_coords, p[0.6868, 0.1598, -0.0020, 0, 0, 0])
    movel(p[new_pose[0], new_pose[1], new_pose[2], current_pose[3], current_pose[4], current_pose[5]], a=0.8, v=0.2000)
    report_progress()
    set_digital_out(0, True)
    new_pose = pose_trans(tuft_coords, p[0.6868, 0.8902, -0.0020, 0, 0, 0])
    movel(p[new_pose[0], new_pose[1], new_pose[2], current_pose[3], current_pose[4], current_pose[5]], a=1.2, v=0.0600)
    report_progress()
    set_digital_out(0, False)
    new_pose = pose_trans(tuft_coords, p[0.6868, 0.8902, 0.1500, 0, 0, 0])
    movel(p[new_pose[0], new_pose[1], new_pose[2], current_pose[3], current_pose[4], current_pose[5]], a=0.8, v=0.2000)
    report_progress()
    new_pose = pose_trans(tuft_coords, p[0.6887, 0.1598, 0.1500, 0, 0, 0])
    movel(p[new_pose[0], new_pose[1], new_pose[2], current_pose[3], current_pose[4], current_pose[5]], a=1.2, v=0.2000)
    report_progress()
    new_pose = pose_trans(tuft_coords, p[0.6887, 0.1598, -0.0020, 0, 0, 0])
    movel(p[new_pose[0], new_pose[1], new_pose[2], current_pose[3], current_pose[4], current_pose[5]], a=0.8, v=0.2000)
    report_progress()
    set_digital_out(0, True)
    new_pose = pose_trans(tuft_coords, p[0.6887, 0.8902, -0.0020, 0, 0, 0])
    movel(p[new_pose[0], new_pose[1], new_pose[2], current_pose[3], current_pose[4], current_pose[5]], a=1.2, v=0.0600)
    report_progress()
    set_digital_out(0, False)
    new_pose = pose_trans(tuft_coords, p[0.6887, 0.8902, 0.1500, 0, 0, 0])
    movel(p[new_pose[0], new_pose[1], new_pose[2], current_pose[3], current_pose[4], current_pose[5]], a=0.8, v=0.2000)
    report_progress()
    new_pose = pose_trans(tuft_coords, p[0.6907, 0.1598, 0.1500, 0, 0, 0])
    movel(p[new_pose[0], new_pose[1], new_pose[2], current_pose[3], current_pose[4], current_pose[5]], a=1.2, v=0.2000)
    report_progress()
    new_pose = pose_trans(tuft_coords, p[0.6907, 0.1598, -0.0020, 0, 0, 0])
    movel(p[new_pose[0], new_pose[1], new_pose[2], current_pose[3], current_pose[4], current_pose[5]], a=0.8, v=0.2000)
    report_progress()
    set_digital_out(0, True)
    new_pose = pose_trans(tuft_coords, p[0.6907, 0.8902, -0.0020, 0, 0, 0])
    movel(p[new_pose[0], new_pose[1], new_pose[2], current_pose[3], current_pose[4], current_pose[5]], a=1.2, v=0.0600)
    report_progress()
    set_digital_out(0, False)
    new_pose = pose_trans(tuft_coords, p[0.6907, 0.8902, 0.1500, 0, 0, 0])
    movel(p[new_pose[0], new_pose[1], new_pose[2], current_pose[3], current_pose[4], current_pose[5]], a=0.8, v=0.2000)
    report_progress()
    new_pose = pose_trans(tuft_coords, p[0.6926, 0.1598, 0.1500, 0, 0, 0])
    movel(p[new_pose[0], new_pose[1], new_pose[2], current_pose[3], current_pose[4], current_pose[5]], a=1.2, v=0.2000)
    report_progress()
    new_pose = pose_trans(tuft_coords, p[0.6926, 0.1598, -0.0020, 0, 0, 0])
    movel(p[new_pose[0], new_pose[1], new_pose[2], current_pose[3], current_pose[4], current_pose[5]], a=0.8, v=0.2000)
    report_progress()
    set_digital_out(0, True)
    new_pose = pose_trans(tuft_coords, p[0.6926, 0.8902, -0.0020, 0, 0, 0])
    movel(p[new_pose[0], new_pose[1], new_pose[2], current_pose[3], current_pose[4], current_pose[5]], a=1.2, v=0.0600)
    report_progress()
    set_digital_out(0, False)
    new_pose = pose_trans(tuft_coords, p[0.6926, 0.8902, 0.1500, 0, 0, 0])
    movel(p[new_pose[0], new_pose[1], new_pose[2], current_pose[3], current_pose[4], current_pose[5]], a=0.8, v=0.2000)
    report_progress()
    new_pose = pose_trans(tuft_coords, p[0.6946, 0.1579, 0.1500, 0, 0, 0])
    movel(p[new_pose[0], new_pose[1], new_pose[2], current_pose[3], current_pose[4], current_pose[5]], a=1.2, v=0.2000)
    report_progress()
    new_pose = pose_trans(tuft_coords, p[0.6946, 0.1579, -0.0020, 0, 0, 0])
    movel(p[new_pose[0], new_pose[1], new_pose[2], current_pose[3], current_pose[4], current_pose[5]], a=0.8, v=0.2000)
    report_progress()
    set_digital_out(0, True)
    new_pose = pose_trans(tuft_coords, p[0.6946, 0.8921, -0.0020, 0, 0, 0])
    movel(p[new_pose[0], new_pose[1], new_pose[2], current_pose[3], current_pose[4], current_pose[5]], a=1.2, v=0.0600)
    report_progress()
    set_digital_out(0, False)
    new_pose = pose_trans(tuft_coords, p[0.6946, 0.8921, 0.1500, 0, 0, 0])
    movel(p[new_pose[0], new_pose[1], new_pose[2], current_pose[3], current_pose[4], current_pose[5]], a=0.8, v=0.2000)
    report_progress()
    new_pose = pose_trans(tuft_coords, p[0.6965, 0.1579, 0.1500, 0, 0, 0])
    movel(p[new_pose[0], new_pose[1], new_pose[2], current_pose[3], current_pose[4], current_pose[5]], a=1.2, v=0.2000)
    report_progress()
    new_pose = pose_trans(tuft_coords, p[0.6965, 0.1579, -0.0020, 0, 0, 0])
    movel(p[new_pose[0], new_pose[1], new_pose[2], current_pose[3], current_pose[4], current_pose[5]], a=0.8, v=0.2000)
    report_progress()
    set_digital_out(0, True)
    new_pose = pose_trans(tuft_coords, p[0.6965, 0.8921, -0.0020, 0, 0, 0])
    movel(p[new_pose[0], new_pose[1], new_pose[2], current_pose[3], current_pose[4], current_pose[5]], a=1.2, v=0.0600)
    report_progress()
    set_digital_out(0, False)
    new_pose = pose_trans(tuft_coords, p[0.6965, 0.8921, 0.1500, 0, 0, 0])
    movel(p[new_pose[0], new_pose[1], new_pose[2], current_pose[3], current_pose[4], current_pose[5]], a=0.8, v=0.2000)
    report_progress()
    new_pose = pose_trans(tuft_coords, p[0.6985, 0.1579, 0.1500, 0, 0, 0])
    movel(p[new_pose[0], new_pose[1], new_pose[2], current_pose[3], current_pose[4], current_pose[5]], a=1.2, v=0.2000)
    report_progress()
    new_pose = pose_trans(tuft_coords, p[0.6985, 0.1579, -0.0020, 0, 0, 0])
    movel(p[new_pose[0], new_pose[1], new_pose[2], current_pose[3], current_pose[4], current_pose[5]], a=0.8, v=0.2000)
    report_progress()
    set_digital_out(0, True)
    new_pose = pose_trans(tuft_coords, p[0.6985, 0.8921, -0.0020, 0, 0, 0])
    movel(p[new_pose[0], new_pose[1], new_pose[2], current_pose[3], current_pose[4], current_pose[5]], a=1.2, v=0.0600)
    report_progress()
    set_digital_out(0, False)
    new_pose = pose_trans(tuft_coords, p[0.6985, 0.8921, 0.1500, 0, 0, 0])
    movel(p[new_pose[0], new_pose[1], new_pose[2], current_pose[3], current_pose[4], current_pose[5]], a=0.8, v=0.2000)
    report_progress()
    new_pose = pose_trans(tuft_coords, p[0.7004, 0.1579, 0.1500, 0, 0, 0])
    movel(p[new_pose[0], new_pose[1], new_pose[2], current_pose[3], current_pose[4], current_pose[5]], a=1.2, v=0.2000)
    report_progress()
    new_pose = pose_trans(tuft_coords, p[0.7004, 0.1579, -0.0020, 0, 0, 0])
    movel(p[new_pose[0], new_pose[1], new_pose[2], current_pose[3], current_pose[4], current_pose[5]], a=0.8, v=0.2000)
    report_progress()
    set_digital_out(0, True)
    new_pose = pose_trans(tuft_coords, p[0.7004, 0.8921, -0.0020, 0, 0, 0])
    movel(p[new_pose[0], new_pose[1], new_pose[2], current_pose[3], current_pose[4], current_pose[5]], a=1.2, v=0.0600)
    report_progress()
    set_digital_out(0, False)
    new_pose = pose_trans(tuft_coords, p[0.7004, 0.8921, 0.1500, 0, 0, 0])
    movel(p[new_pose[0], new_pose[1], new_pose[2], current_pose[3], current_pose[4], current_pose[5]], a=0.8, v=0.2000)
    report_progress()
    new_pose = pose_trans(tuft_coords, p[0.7024, 0.1579, 0.1500, 0, 0, 0])
    movel(p[new_pose[0], new_pose[1], new_pose[2], current_pose[3], current_pose[4], current_pose[5]], a=1.2, v=0.2000)
    report_progress()
    new_pose = pose_trans(tuft_coords, p[0.7024, 0.1579, -0.0020, 0, 0, 0])
    movel(p[new_pose[0], new_pose[1], new_pose[2], current_pose[3], current_pose[4], current_pose[5]], a=0.8, v=0.2000)
    report_progress()
    set_digital_out(0, True)
    new_pose = pose_trans(tuft_coords, p[0.7024, 0.8921, -0.0020, 0, 0, 0])
    movel(p[new_pose[0], new_pose[1], new_pose[2], current_pose[3], current_pose[4], current_pose[5]], a=1.2, v=0.0600)
    report_progress()
    set_digital_out(0, False)
    new_pose = pose_trans(tuft_coords, p[0.7024, 0.8921, 0.1500, 0, 0, 0])
    movel(p[new_pose[0], new_pose[1], new_pose[2], current_pose[3], current_pose[4], current_pose[5]], a=0.8, v=0.2000)
    report_progress()
    new_pose = pose_trans(tuft_coords, p[0.7043, 0.1579, 0.1500, 0, 0, 0])
    movel(p[new_pose[0], new_pose[1], new_pose[2], current_pose[3], current_pose[4], current_pose[5]], a=1.2, v=0.2000)
    report_progress()
    new_pose = pose_trans(tuft_coords, p[0.7043, 0.1579, -0.0020, 0, 0, 0])
    movel(p[new_pose[0], new_pose[1], new_pose[2], current_pose[3], current_pose[4], current_pose[5]], a=0.8, v=0.2000)
    report_progress()
    set_digital_out(0, True)
    new_pose = pose_trans(tuft_coords, p[0.7043, 0.8921, -0.0020, 0, 0, 0])
    movel(p[new_pose[0], new_pose[1], new_pose[2], current_pose[3], current_pose[4], current_pose[5]], a=1.2, v=0.0600)
    report_progress()
    set_digital_out(0, False)
    new_pose = pose_trans(tuft_coords, p[0.7043, 0.8921, 0.1500, 0, 0, 0])
    movel(p[new_pose[0], new_pose[1], new_pose[2], current_pose[3], current_pose[4], current_pose[5]], a=0.8, v=0.2000)
    report_progress()
    new_pose = pose_trans(tuft_coords, p[0.7063, 0.1579, 0.1500, 0, 0, 0])
    movel(p[new_pose[0], new_pose[1], new_pose[2], current_pose[3], current_pose[4], current_pose[5]], a=1.2, v=0.2000)
    report_progress()
    new_pose = pose_trans(tuft_coords, p[0.7063, 0.1579, -0.0020, 0, 0, 0])
    movel(p[new_pose[0], new_pose[1], new_pose[2], current_pose[3], current_pose[4], current_pose[5]], a=0.8, v=0.2000)
    report_progress()
    set_digital_out(0, True)
    new_pose = pose_trans(tuft_coords, p[0.7063, 0.8921, -0.0020, 0, 0, 0])
    movel(p[new_pose[0], new_pose[1], new_pose[2], current_pose[3], current_pose[4], current_pose[5]], a=1.2, v=0.0600)
    report_progress()
    set_digital_out(0, False)
    new_pose = pose_trans(tuft_coords, p[0.7063, 0.8921, 0.1500, 0, 0, 0])
    movel(p[new_pose[0], new_pose[1], new_pose[2], current_pose[3], current_pose[4], current_pose[5]], a=0.8, v=0.2000)
    report_progress()
    new_pose = pose_trans(tuft_coords, p[0.7082, 0.1559, 0.1500, 0, 0, 0])
    movel(p[new_pose[0], new_pose[1], new_pose[2], current_pose[3], current_pose[4], current_pose[5]], a=1.2, v=0.2000)
    report_progress()
    new_pose = pose_trans(tuft_coords, p[0.7082, 0.1559, -0.0020, 0, 0, 0])
    movel(p[new_pose[0], new_pose[1], new_pose[2], current_pose[3], current_pose[4], current_pose[5]], a=0.8, v=0.2000)
    report_progress()
    set_digital_out(0, True)
    new_pose = pose_trans(tuft_coords, p[0.7082, 0.8941, -0.0020, 0, 0, 0])
    movel(p[new_pose[0], new_pose[1], new_pose[2], current_pose[3], current_pose[4], current_pose[5]], a=1.2, v=0.0600)
    report_progress()
    set_digital_out(0, False)
    new_pose = pose_trans(tuft_coords, p[0.7082, 0.8941, 0.1500, 0, 0, 0])
    movel(p[new_pose[0], new_pose[1], new_pose[2], current_pose[3], current_pose[4], current_pose[5]], a=0.8, v=0.2000)
    report_progress()
    new_pose = pose_trans(tuft_coords, p[0.7101, 0.1559, 0.1500, 0, 0, 0])
    movel(p[new_pose[0], new_pose[1], new_pose[2], current_pose[3], current_pose[4], current_pose[5]], a=1.2, v=0.2000)
    report_progress()
    new_pose = pose_trans(tuft_coords, p[0.7101, 0.1559, -0.0020, 0, 0, 0])
    movel(p[new_pose[0], new_pose[1], new_pose[2], current_pose[3], current_pose[4], current_pose[5]], a=0.8, v=0.2000)
    report_progress()
    set_digital_out(0, True)
    new_pose = pose_trans(tuft_coords, p[0.7101, 0.8941, -0.0020, 0, 0, 0])
    movel(p[new_pose[0], new_pose[1], new_pose[2], current_pose[3], current_pose[4], current_pose[5]], a=1.2, v=0.0600)
    report_progress()
    set_digital_out(0, False)
    new_pose = pose_trans(tuft_coords, p[0.7101, 0.8941, 0.1500, 0, 0, 0])
    movel(p[new_pose[0], new_pose[1], new_pose[2], current_pose[3], current_pose[4], current_pose[5]], a=0.8, v=0.2000)
    report_progress()
    new_pose = pose_trans(tuft_coords, p[0.7121, 0.1559, 0.1500, 0, 0, 0])
    movel(p[new_pose[0], new_pose[1], new_pose[2], current_pose[3], current_pose[4], current_pose[5]], a=1.2, v=0.2000)
    report_progress()
    new_pose = pose_trans(tuft_coords, p[0.7121, 0.1559, -0.0020, 0, 0, 0])
    movel(p[new_pose[0], new_pose[1], new_pose[2], current_pose[3], current_pose[4], current_pose[5]], a=0.8, v=0.2000)
    report_progress()
    set_digital_out(0, True)
    new_pose = pose_trans(tuft_coords, p[0.7121, 0.8941, -0.0020, 0, 0, 0])
    movel(p[new_pose[0], new_pose[1], new_pose[2], current_pose[3], current_pose[4], current_pose[5]], a=1.2, v=0.0600)
    report_progress()
    set_digital_out(0, False)
    new_pose = pose_trans(tuft_coords, p[0.7121, 0.8941, 0.1500, 0, 0, 0])
    movel(p[new_pose[0], new_pose[1], new_pose[2], current_pose[3], current_pose[4], current_pose[5]], a=0.8, v=0.2000)
    report_progress()
    new_pose = pose_trans(tuft_coords, p[0.7140, 0.1559, 0.1500, 0, 0, 0])
    movel(p[new_pose[0], new_pose[1], new_pose[2], current_pose[3], current_pose[4], current_pose[5]], a=1.2, v=0.2000)
    report_progress()
    new_pose = pose_trans(tuft_coords, p[0.7140, 0.1559, -0.0020, 0, 0, 0])
    movel(p[new_pose[0], new_pose[1], new_pose[2], current_pose[3], current_pose[4], current_pose[5]], a=0.8, v=0.2000)
    report_progress()
    set_digital_out(0, True)
    new_pose = pose_trans(tuft_coords, p[0.7140, 0.8941, -0.0020, 0, 0, 0])
    movel(p[new_pose[0], new_pose[1], new_pose[2], current_pose[3], current_pose[4], current_pose[5]], a=1.2, v=0.0600)
    report_progress()
    set_digital_out(0, False)
    new_pose = pose_trans(tuft_coords, p[0.7140, 0.8941, 0.1500, 0, 0, 0])
    movel(p[new_pose[0], new_pose[1], new_pose[2], current_pose[3], current_pose[4], current_pose[5]], a=0.8, v=0.2000)
    report_progress()
    new_pose = pose_trans(tuft_coords, p[0.7160, 0.1559, 0.1500, 0, 0, 0])
    movel(p[new_pose[0], new_pose[1], new_pose[2], current_pose[3], current_pose[4], current_pose[5]], a=1.2, v=0.2000)
    report_progress()
    new_pose = pose_trans(tuft_coords, p[0.7160, 0.1559, -0.0020, 0, 0, 0])
    movel(p[new_pose[0], new_pose[1], new_pose[2], current_pose[3], current_pose[4], current_pose[5]], a=0.8, v=0.2000)
    report_progress()
    set_digital_out(0, True)
    new_pose = pose_trans(tuft_coords, p[0.7160, 0.8941, -0.0020, 0, 0, 0])
    movel(p[new_pose[0], new_pose[1], new_pose[2], current_pose[3], current_pose[4], current_pose[5]], a=1.2, v=0.0600)
    report_progress()
    set_digital_out(0, False)
    new_pose = pose_trans(tuft_coords, p[0.7160, 0.8941, 0.1500, 0, 0, 0])
    movel(p[new_pose[0], new_pose[1], new_pose[2], current_pose[3], current_pose[4], current_pose[5]], a=0.8, v=0.2000)
    report_progress()
    new_pose = pose_trans(tuft_coords, p[0.7179, 0.1559, 0.1500, 0, 0, 0])
    movel(p[new_pose[0], new_pose[1], new_pose[2], current_pose[3], current_pose[4], current_pose[5]], a=1.2, v=0.2000)
    report_progress()
    new_pose = pose_trans(tuft_coords, p[0.7179, 0.1559, -0.0020, 0, 0, 0])
    movel(p[new_pose[0], new_pose[1], new_pose[2], current_pose[3], current_pose[4], current_pose[5]], a=0.8, v=0.2000)
    report_progress()
    set_digital_out(0, True)
    new_pose = pose_trans(tuft_coords, p[0.7179, 0.8941, -0.0020, 0, 0, 0])
    movel(p[new_pose[0], new_pose[1], new_pose[2], current_pose[3], current_pose[4], current_pose[5]], a=1.2, v=0.0600)
    report_progress()
    set_digital_out(0, False)
    new_pose = pose_trans(tuft_coords, p[0.7179, 0.8941, 0.1500, 0, 0, 0])
    movel(p[new_pose[0], new_pose[1], new_pose[2], current_pose[3], current_pose[4], current_pose[5]], a=0.8, v=0.2000)
    report_progress()
    new_pose = pose_trans(tuft_coords, p[0.7199, 0.1559, 0.1500, 0, 0, 0])
    movel(p[new_pose[0], new_pose[1], new_pose[2], current_pose[3], current_pose[4], current_pose[5]], a=1.2, v=0.2000)
    report_progress()
    new_pose = pose_trans(tuft_coords, p[0.7199, 0.1559, -0.0020, 0, 0, 0])
    movel(p[new_pose[0], new_pose[1], new_pose[2], current_pose[3], current_pose[4], current_pose[5]], a=0.8, v=0.2000)
    report_progress()
    set_digital_out(0, True)
    new_pose = pose_trans(tuft_coords, p[0.7199, 0.8941, -0.0020, 0, 0, 0])
    movel(p[new_pose[0], new_pose[1], new_pose[2], current_pose[3], current_pose[4], current_pose[5]], a=1.2, v=0.0600)
    report_progress()
    set_digital_out(0, False)
    new_pose = pose_trans(tuft_coords, p[0.7199, 0.8941, 0.1500, 0, 0, 0])
    movel(p[new_pose[0], new_pose[1], new_pose[2], current_pose[3], current_pose[4], current_pose[5]], a=0.8, v=0.2000)
    report_progress()
    new_pose = pose_trans(tuft_coords, p[0.7218, 0.1559, 0.1500, 0, 0, 0])
    movel(p[new_pose[0], new_pose[1], new_pose[2], current_pose[3], current_pose[4], current_pose[5]], a=1.2, v=0.2000)
    report_progress()
    new_pose = pose_trans(tuft_coords, p[0.7218, 0.1559, -0.0020, 0, 0, 0])
    movel(p[new_pose[0], new_pose[1], new_pose[2], current_pose[3], current_pose[4], current_pose[5]], a=0.8, v=0.2000)
    report_progress()
    set_digital_out(0, True)
    new_pose = pose_trans(tuft_coords, p[0.7218, 0.8941, -0.0020, 0, 0, 0])
    movel(p[new_pose[0], new_pose[1], new_pose[2], current_pose[3], current_pose[4], current_pose[5]], a=1.2, v=0.0600)
    report_progress()
    set_digital_out(0, False)
    new_pose = pose_trans(tuft_coords, p[0.7218, 0.8941, 0.1500, 0, 0, 0])
    movel(p[new_pose[0], new_pose[1], new_pose[2], current_pose[3], current_pose[4], current_pose[5]], a=0.8, v=0.2000)
    report_progress()
    new_pose = pose_trans(tuft_coords, p[0.7238, 0.1559, 0.1500, 0, 0, 0])
    movel(p[new_pose[0], new_pose[1], new_pose[2], current_pose[3], current_pose[4], current_pose[5]], a=1.2, v=0.2000)
    report_progress()
    new_pose = pose_trans(tuft_coords, p[0.7238, 0.1559, -0.0020, 0, 0, 0])
    movel(p[new_pose[0], new_pose[1], new_pose[2], current_pose[3], current_pose[4], current_pose[5]], a=0.8, v=0.2000)
    report_progress()
    set_digital_out(0, True)
    new_pose = pose_trans(tuft_coords, p[0.7238, 0.8941, -0.0020, 0, 0, 0])
    movel(p[new_pose[0], new_pose[1], new_pose[2], current_pose[3], current_pose[4], current_pose[5]], a=1.2, v=0.0600)
    report_progress()
    set_digital_out(0, False)
    new_pose = pose_trans(tuft_coords, p[0.7238, 0.8941, 0.1500, 0, 0, 0])
    movel(p[new_pose[0], new_pose[1], new_pose[2], current_pose[3], current_pose[4], current_pose[5]], a=0.8, v=0.2000)
    report_progress()
    new_pose = pose_trans(tuft_coords, p[0.7257, 0.1559, 0.1500, 0, 0, 0])
    movel(p[new_pose[0], new_pose[1], new_pose[2], current_pose[3], current_pose[4], current_pose[5]], a=1.2, v=0.2000)
    report_progress()
    new_pose = pose_trans(tuft_coords, p[0.7257, 0.1559, -0.0020, 0, 0, 0])
    movel(p[new_pose[0], new_pose[1], new_pose[2], current_pose[3], current_pose[4], current_pose[5]], a=0.8, v=0.2000)
    report_progress()
    set_digital_out(0, True)
    new_pose = pose_trans(tuft_coords, p[0.7257, 0.8941, -0.0020, 0, 0, 0])
    movel(p[new_pose[0], new_pose[1], new_pose[2], current_pose[3], current_pose[4], current_pose[5]], a=1.2, v=0.0600)
    report_progress()
    set_digital_out(0, False)
    new_pose = pose_trans(tuft_coords, p[0.7257, 0.8941, 0.1500, 0, 0, 0])
    movel(p[new_pose[0], new_pose[1], new_pose[2], current_pose[3], current_pose[4], current_pose[5]], a=0.8, v=0.2000)
    report_progress()
    new_pose = pose_trans(tuft_coords, p[0.7276, 0.1559, 0.1500, 0, 0, 0])
    movel(p[new_pose[0], new_pose[1], new_pose[2], current_pose[3], current_pose[4], current_pose[5]], a=1.2, v=0.2000)
    report_progress()
    new_pose = pose_trans(tuft_coords, p[0.7276, 0.1559, -0.0020, 0, 0, 0])
    movel(p[new_pose[0], new_pose[1], new_pose[2], current_pose[3], current_pose[4], current_pose[5]], a=0.8, v=0.2000)
    report_progress()
    set_digital_out(0, True)
    new_pose = pose_trans(tuft_coords, p[0.7276, 0.8941, -0.0020, 0, 0, 0])
    movel(p[new_pose[0], new_pose[1], new_pose[2], current_pose[3], current_pose[4], current_pose[5]], a=1.2, v=0.0600)
    report_progress()
    set_digital_out(0, False)
    new_pose = pose_trans(tuft_coords, p[0.7276, 0.8941, 0.1500, 0, 0, 0])
    movel(p[new_pose[0], new_pose[1], new_pose[2], current_pose[3], current_pose[4], current_pose[5]], a=0.8, v=0.2000)
    report_progress()
    new_pose = pose_trans(tuft_coords, p[0.7296, 0.1559, 0.1500, 0, 0, 0])
    movel(p[new_pose[0], new_pose[1], new_pose[2], current_pose[3], current_pose[4], current_pose[5]], a=1.2, v=0.2000)
    report_progress()
    new_pose = pose_trans(tuft_coords, p[0.7296, 0.1559, -0.0020, 0, 0, 0])
    movel(p[new_pose[0], new_pose[1], new_pose[2], current_pose[3], current_pose[4], current_pose[5]], a=0.8, v=0.2000)
    report_progress()
    set_digital_out(0, True)
    new_pose = pose_trans(tuft_coords, p[0.7296, 0.8941, -0.0020, 0, 0, 0])
    movel(p[new_pose[0], new_pose[1], new_pose[2], current_pose[3], current_pose[4], current_pose[5]], a=1.2, v=0.0600)
    report_progress()
    set_digital_out(0, False)
    new_pose = pose_trans(tuft_coords, p[0.7296, 0.8941, 0.1500, 0, 0, 0])
    movel(p[new_pose[0], new_pose[1], new_pose[2], current_pose[3], current_pose[4], current_pose[5]], a=0.8, v=0.2000)
    report_progress()
    new_pose = pose_trans(tuft_coords, p[0.7315, 0.1539, 0.1500, 0, 0, 0])
    movel(p[new_pose[0], new_pose[1], new_pose[2], current_pose[3], current_pose[4], current_pose[5]], a=1.2, v=0.2000)
    report_progress()
    new_pose = pose_trans(tuft_coords, p[0.7315, 0.1539, -0.0020, 0, 0, 0])
    movel(p[new_pose[0], new_pose[1], new_pose[2], current_pose[3], current_pose[4], current_pose[5]], a=0.8, v=0.2000)
    report_progress()
    set_digital_out(0, True)
    new_pose = pose_trans(tuft_coords, p[0.7315, 0.8961, -0.0020, 0, 0, 0])
    movel(p[new_pose[0], new_pose[1], new_pose[2], current_pose[3], current_pose[4], current_pose[5]], a=1.2, v=0.0600)
    report_progress()
    set_digital_out(0, False)
    new_pose = pose_trans(tuft_coords, p[0.7315, 0.8961, 0.1500, 0, 0, 0])
    movel(p[new_pose[0], new_pose[1], new_pose[2], current_pose[3], current_pose[4], current_pose[5]], a=0.8, v=0.2000)
    report_progress()
    new_pose = pose_trans(tuft_coords, p[0.7335, 0.1539, 0.1500, 0, 0, 0])
    movel(p[new_pose[0], new_pose[1], new_pose[2], current_pose[3], current_pose[4], current_pose[5]], a=1.2, v=0.2000)
    report_progress()
    new_pose = pose_trans(tuft_coords, p[0.7335, 0.1539, -0.0020, 0, 0, 0])
    movel(p[new_pose[0], new_pose[1], new_pose[2], current_pose[3], current_pose[4], current_pose[5]], a=0.8, v=0.2000)
    report_progress()
    set_digital_out(0, True)
    new_pose = pose_trans(tuft_coords, p[0.7335, 0.8961, -0.0020, 0, 0, 0])
    movel(p[new_pose[0], new_pose[1], new_pose[2], current_pose[3], current_pose[4], current_pose[5]], a=1.2, v=0.0600)
    report_progress()
    set_digital_out(0, False)
    new_pose = pose_trans(tuft_coords, p[0.7335, 0.8961, 0.1500, 0, 0, 0])
    movel(p[new_pose[0], new_pose[1], new_pose[2], current_pose[3], current_pose[4], current_pose[5]], a=0.8, v=0.2000)
    report_progress()
    new_pose = pose_trans(tuft_coords, p[0.7354, 0.1539, 0.1500, 0, 0, 0])
    movel(p[new_pose[0], new_pose[1], new_pose[2], current_pose[3], current_pose[4], current_pose[5]], a=1.2, v=0.2000)
    report_progress()
    new_pose = pose_trans(tuft_coords, p[0.7354, 0.1539, -0.0020, 0, 0, 0])
    movel(p[new_pose[0], new_pose[1], new_pose[2], current_pose[3], current_pose[4], current_pose[5]], a=0.8, v=0.2000)
    report_progress()
    set_digital_out(0, True)
    new_pose = pose_trans(tuft_coords, p[0.7354, 0.8961, -0.0020, 0, 0, 0])
    movel(p[new_pose[0], new_pose[1], new_pose[2], current_pose[3], current_pose[4], current_pose[5]], a=1.2, v=0.0600)
    report_progress()
    set_digital_out(0, False)
    new_pose = pose_trans(tuft_coords, p[0.7354, 0.8961, 0.1500, 0, 0, 0])
    movel(p[new_pose[0], new_pose[1], new_pose[2], current_pose[3], current_pose[4], current_pose[5]], a=0.8, v=0.2000)
    report_progress()
    new_pose = pose_trans(tuft_coords, p[0.7374, 0.1539, 0.1500, 0, 0, 0])
    movel(p[new_pose[0], new_pose[1], new_pose[2], current_pose[3], current_pose[4], current_pose[5]], a=1.2, v=0.2000)
    report_progress()
    new_pose = pose_trans(tuft_coords, p[0.7374, 0.1539, -0.0020, 0, 0, 0])
    movel(p[new_pose[0], new_pose[1], new_pose[2], current_pose[3], current_pose[4], current_pose[5]], a=0.8, v=0.2000)
    report_progress()
    set_digital_out(0, True)
    new_pose = pose_trans(tuft_coords, p[0.7374, 0.8961, -0.0020, 0, 0, 0])
    movel(p[new_pose[0], new_pose[1], new_pose[2], current_pose[3], current_pose[4], current_pose[5]], a=1.2, v=0.0600)
    report_progress()
    set_digital_out(0, False)
    new_pose = pose_trans(tuft_coords, p[0.7374, 0.8961, 0.1500, 0, 0, 0])
    movel(p[new_pose[0], new_pose[1], new_pose[2], current_pose[3], current_pose[4], current_pose[5]], a=0.8, v=0.2000)
    report_progress()
    new_pose = pose_trans(tuft_coords, p[0.7393, 0.1539, 0.1500, 0, 0, 0])
    movel(p[new_pose[0], new_pose[1], new_pose[2], current_pose[3], current_pose[4], current_pose[5]], a=1.2, v=0.2000)
    report_progress()
    new_pose = pose_trans(tuft_coords, p[0.7393, 0.1539, -0.0020, 0, 0, 0])
    movel(p[new_pose[0], new_pose[1], new_pose[2], current_pose[3], current_pose[4], current_pose[5]], a=0.8, v=0.2000)
    report_progress()
    set_digital_out(0, True)
    new_pose = pose_trans(tuft_coords, p[0.7393, 0.8961, -0.0020, 0, 0, 0])
    movel(p[new_pose[0], new_pose[1], new_pose[2], current_pose[3], current_pose[4], current_pose[5]], a=1.2, v=0.0600)
    report_progress()
    set_digital_out(0, False)
    new_pose = pose_trans(tuft_coords, p[0.7393, 0.8961, 0.1500, 0, 0, 0])
    movel(p[new_pose[0], new_pose[1], new_pose[2], current_pose[3], current_pose[4], current_pose[5]], a=0.8, v=0.2000)
    report_progress()
    new_pose = pose_trans(tuft_coords, p[0.7412, 0.1539, 0.1500, 0, 0, 0])
    movel(p[new_pose[0], new_pose[1], new_pose[2], current_pose[3], current_pose[4], current_pose[5]], a=1.2, v=0.2000)
    report_progress()
    new_pose = pose_trans(tuft_coords, p[0.7412, 0.1539, -0.0020, 0, 0, 0])
    movel(p[new_pose[0], new_pose[1], new_pose[2], current_pose[3], current_pose[4], current_pose[5]], a=0.8, v=0.2000)
    report_progress()
    set_digital_out(0, True)
    new_pose = pose_trans(tuft_coords, p[0.7412, 0.8961, -0.0020, 0, 0, 0])
    movel(p[new_pose[0], new_pose[1], new_pose[2], current_pose[3], current_pose[4], current_pose[5]], a=1.2, v=0.0600)
    report_progress()
    set_digital_out(0, False)
    new_pose = pose_trans(tuft_coords, p[0.7412, 0.8961, 0.1500, 0, 0, 0])
    movel(p[new_pose[0], new_pose[1], new_pose[2], current_pose[3], current_pose[4], current_pose[5]], a=0.8, v=0.2000)
    report_progress()
    new_pose = pose_trans(tuft_coords, p[0.7432, 0.1539, 0.1500, 0, 0, 0])
    movel(p[new_pose[0], new_pose[1], new_pose[2], current_pose[3], current_pose[4], current_pose[5]], a=1.2, v=0.2000)
    report_progress()
    new_pose = pose_trans(tuft_coords, p[0.7432, 0.1539, -0.0020, 0, 0, 0])
    movel(p[new_pose[0], new_pose[1], new_pose[2], current_pose[3], current_pose[4], current_pose[5]], a=0.8, v=0.2000)
    report_progress()
    set_digital_out(0, True)
    new_pose = pose_trans(tuft_coords, p[0.7432, 0.8961, -0.0020, 0, 0, 0])
    movel(p[new_pose[0], new_pose[1], new_pose[2], current_pose[3], current_pose[4], current_pose[5]], a=1.2, v=0.0600)
    report_progress()
    set_digital_out(0, False)
    new_pose = pose_trans(tuft_coords, p[0.7432, 0.8961, 0.1500, 0, 0, 0])
    movel(p[new_pose[0], new_pose[1], new_pose[2], current_pose[3], current_pose[4], current_pose[5]], a=0.8, v=0.2000)
    report_progress()
    new_pose = pose_trans(tuft_coords, p[0.7451, 0.1539, 0.1500, 0, 0, 0])
    movel(p[new_pose[0], new_pose[1], new_pose[2], current_pose[3], current_pose[4], current_pose[5]], a=1.2, v=0.2000)
    report_progress()
    new_pose = pose_trans(tuft_coords, p[0.7451, 0.1539, -0.0020, 0, 0, 0])
    movel(p[new_pose[0], new_pose[1], new_pose[2], current_pose[3], current_pose[4], current_pose[5]], a=0.8, v=0.2000)
    report_progress()
    set_digital_out(0, True)
    new_pose = pose_trans(tuft_coords, p[0.7451, 0.8961, -0.0020, 0, 0, 0])
    movel(p[new_pose[0], new_pose[1], new_pose[2], current_pose[3], current_pose[4], current_pose[5]], a=1.2, v=0.0600)
    report_progress()
    set_digital_out(0, False)
    new_pose = pose_trans(tuft_coords, p[0.7451, 0.8961, 0.1500, 0, 0, 0])
    movel(p[new_pose[0], new_pose[1], new_pose[2], current_pose[3], current_pose[4], current_pose[5]], a=0.8, v=0.2000)
    report_progress()
    new_pose = pose_trans(tuft_coords, p[0.7471, 0.1539, 0.1500, 0, 0, 0])
    movel(p[new_pose[0], new_pose[1], new_pose[2], current_pose[3], current_pose[4], current_pose[5]], a=1.2, v=0.2000)
    report_progress()
    new_pose = pose_trans(tuft_coords, p[0.7471, 0.1539, -0.0020, 0, 0, 0])
    movel(p[new_pose[0], new_pose[1], new_pose[2], current_pose[3], current_pose[4], current_pose[5]], a=0.8, v=0.2000)
    report_progress()
    set_digital_out(0, True)
    new_pose = pose_trans(tuft_coords, p[0.7471, 0.8961, -0.0020, 0, 0, 0])
    movel(p[new_pose[0], new_pose[1], new_pose[2], current_pose[3], current_pose[4], current_pose[5]], a=1.2, v=0.0600)
    report_progress()
    set_digital_out(0, False)
    new_pose = pose_trans(tuft_coords, p[0.7471, 0.8961, 0.1500, 0, 0, 0])
    movel(p[new_pose[0], new_pose[1], new_pose[2], current_pose[3], current_pose[4], current_pose[5]], a=0.8, v=0.2000)
    report_progress()
    new_pose = pose_trans(tuft_coords, p[0.7490, 0.1539, 0.1500, 0, 0, 0])
    movel(p[new_pose[0], new_pose[1], new_pose[2], current_pose[3], current_pose[4], current_pose[5]], a=1.2, v=0.2000)
    report_progress()
    new_pose = pose_trans(tuft_coords, p[0.7490, 0.1539, -0.0020, 0, 0, 0])
    movel(p[new_pose[0], new_pose[1], new_pose[2], current_pose[3], current_pose[4], current_pose[5]], a=0.8, v=0.2000)
    report_progress()
    set_digital_out(0, True)
    new_pose = pose_trans(tuft_coords, p[0.7490, 0.8961, -0.0020, 0, 0, 0])
    movel(p[new_pose[0], new_pose[1], new_pose[2], current_pose[3], current_pose[4], current_pose[5]], a=1.2, v=0.0600)
    report_progress()
    set_digital_out(0, False)
    new_pose = pose_trans(tuft_coords, p[0.7490, 0.8961, 0.1500, 0, 0, 0])
    movel(p[new_pose[0], new_pose[1], new_pose[2], current_pose[3], current_pose[4], current_pose[5]], a=0.8, v=0.2000)
    report_progress()
    new_pose = pose_trans(tuft_coords, p[0.7510, 0.1539, 0.1500, 0, 0, 0])
    movel(p[new_pose[0], new_pose[1], new_pose[2], current_pose[3], current_pose[4], current_pose[5]], a=1.2, v=0.2000)
    report_progress()
    new_pose = pose_trans(tuft_coords, p[0.7510, 0.1539, -0.0020, 0, 0, 0])
    movel(p[new_pose[0], new_pose[1], new_pose[2], current_pose[3], current_pose[4], current_pose[5]], a=0.8, v=0.2000)
    report_progress()
    set_digital_out(0, True)
    new_pose = pose_trans(tuft_coords, p[0.7510, 0.8961, -0.0020, 0, 0, 0])
    movel(p[new_pose[0], new_pose[1], new_pose[2], current_pose[3], current_pose[4], current_pose[5]], a=1.2, v=0.0600)
    report_progress()
    set_digital_out(0, False)
    new_pose = pose_trans(tuft_coords, p[0.7510, 0.8961, 0.1500, 0, 0, 0])
    movel(p[new_pose[0], new_pose[1], new_pose[2], current_pose[3], current_pose[4], current_pose[5]], a=0.8, v=0.2000)
    report_progress()
    new_pose = pose_trans(tuft_coords, p[0.7529, 0.1539, 0.1500, 0, 0, 0])
    movel(p[new_pose[0], new_pose[1], new_pose[2], current_pose[3], current_pose[4], current_pose[5]], a=1.2, v=0.2000)
    report_progress()
    new_pose = pose_trans(tuft_coords, p[0.7529, 0.1539, -0.0020, 0, 0, 0])
    movel(p[new_pose[0], new_pose[1], new_pose[2], current_pose[3], current_pose[4], current_pose[5]], a=0.8, v=0.2000)
    report_progress()
    set_digital_out(0, True)
    new_pose = pose_trans(tuft_coords, p[0.7529, 0.8961, -0.0020, 0, 0, 0])
    movel(p[new_pose[0], new_pose[1], new_pose[2], current_pose[3], current_pose[4], current_pose[5]], a=1.2, v=0.0600)
    report_progress()
    set_digital_out(0, False)
    new_pose = pose_trans(tuft_coords, p[0.7529, 0.8961, 0.1500, 0, 0, 0])
    movel(p[new_pose[0], new_pose[1], new_pose[2], current_pose[3], current_pose[4], current_pose[5]], a=0.8, v=0.2000)
    report_progress()
    new_pose = pose_trans(tuft_coords, p[0.7549, 0.1539, 0.1500, 0, 0, 0])
    movel(p[new_pose[0], new_pose[1], new_pose[2], current_pose[3], current_pose[4], current_pose[5]], a=1.2, v=0.2000)
    report_progress()
    new_pose = pose_trans(tuft_coords, p[0.7549, 0.1539, -0.0020, 0, 0, 0])
    movel(p[new_pose[0], new_pose[1], new_pose[2], current_pose[3], current_pose[4], current_pose[5]], a=0.8, v=0.2000)
    report_progress()
    set_digital_out(0, True)
    new_pose = pose_trans(tuft_coords, p[0.7549, 0.8961, -0.0020, 0, 0, 0])
    movel(p[new_pose[0], new_pose[1], new_pose[2], current_pose[3], current_pose[4], current_pose[5]], a=1.2, v=0.0600)
    report_progress()
    set_digital_out(0, False)
    new_pose = pose_trans(tuft_coords, p[0.7549, 0.8961, 0.1500, 0, 0, 0])
    movel(p[new_pose[0], new_pose[1], new_pose[2], current_pose[3], current_pose[4], current_pose[5]], a=0.8, v=0.2000)
    report_progress()
    new_pose = pose_trans(tuft_coords, p[0.7568, 0.1539, 0.1500, 0, 0, 0])
    movel(p[new_pose[0], new_pose[1], new_pose[2], current_pose[3], current_pose[4], current_pose[5]], a=1.2, v=0.2000)
    report_progress()
    new_pose = pose_trans(tuft_coords, p[0.7568, 0.1539, -0.0020, 0, 0, 0])
    movel(p[new_pose[0], new_pose[1], new_pose[2], current_pose[3], current_pose[4], current_pose[5]], a=0.8, v=0.2000)
    report_progress()
    set_digital_out(0, True)
    new_pose = pose_trans(tuft_coords, p[0.7568, 0.8961, -0.0020, 0, 0, 0])
    movel(p[new_pose[0], new_pose[1], new_pose[2], current_pose[3], current_pose[4], current_pose[5]], a=1.2, v=0.0600)
    report_progress()
    set_digital_out(0, False)
    new_pose = pose_trans(tuft_coords, p[0.7568, 0.8961, 0.1500, 0, 0, 0])
    movel(p[new_pose[0], new_pose[1], new_pose[2], current_pose[3], current_pose[4], current_pose[5]], a=0.8, v=0.2000)
    report_progress()
    new_pose = pose_trans(tuft_coords, p[0.7588, 0.1539, 0.1500, 0, 0, 0])
    movel(p[new_pose[0], new_pose[1], new_pose[2], current_pose[3], current_pose[4], current_pose[5]], a=1.2, v=0.2000)
    report_progress()
    new_pose = pose_trans(tuft_coords, p[0.7588, 0.1539, -0.0020, 0, 0, 0])
    movel(p[new_pose[0], new_pose[1], new_pose[2], current_pose[3], current_pose[4], current_pose[5]], a=0.8, v=0.2000)
    report_progress()
    set_digital_out(0, True)
    new_pose = pose_trans(tuft_coords, p[0.7588, 0.8961, -0.0020, 0, 0, 0])
    movel(p[new_pose[0], new_pose[1], new_pose[2], current_pose[3], current_pose[4], current_pose[5]], a=1.2, v=0.0600)
    report_progress()
    set_digital_out(0, False)
    new_pose = pose_trans(tuft_coords, p[0.7588, 0.8961, 0.1500, 0, 0, 0])
    movel(p[new_pose[0], new_pose[1], new_pose[2], current_pose[3], current_pose[4], current_pose[5]], a=0.8, v=0.2000)
    report_progress()
    new_pose = pose_trans(tuft_coords, p[0.7607, 0.1539, 0.1500, 0, 0, 0])
    movel(p[new_pose[0], new_pose[1], new_pose[2], current_pose[3], current_pose[4], current_pose[5]], a=1.2, v=0.2000)
    report_progress()
    new_pose = pose_trans(tuft_coords, p[0.7607, 0.1539, -0.0020, 0, 0, 0])
    movel(p[new_pose[0], new_pose[1], new_pose[2], current_pose[3], current_pose[4], current_pose[5]], a=0.8, v=0.2000)
    report_progress()
    set_digital_out(0, True)
    new_pose = pose_trans(tuft_coords, p[0.7607, 0.8961, -0.0020, 0, 0, 0])
    movel(p[new_pose[0], new_pose[1], new_pose[2], current_pose[3], current_pose[4], current_pose[5]], a=1.2, v=0.0600)
    report_progress()
    set_digital_out(0, False)
    new_pose = pose_trans(tuft_coords, p[0.7607, 0.8961, 0.1500, 0, 0, 0])
    movel(p[new_pose[0], new_pose[1], new_pose[2], current_pose[3], current_pose[4], current_pose[5]], a=0.8, v=0.2000)
    report_progress()
    new_pose = pose_trans(tuft_coords, p[0.7626, 0.1539, 0.1500, 0, 0, 0])
    movel(p[new_pose[0], new_pose[1], new_pose[2], current_pose[3], current_pose[4], current_pose[5]], a=1.2, v=0.2000)
    report_progress()
    new_pose = pose_trans(tuft_coords, p[0.7626, 0.1539, -0.0020, 0, 0, 0])
    movel(p[new_pose[0], new_pose[1], new_pose[2], current_pose[3], current_pose[4], current_pose[5]], a=0.8, v=0.2000)
    report_progress()
    set_digital_out(0, True)
    new_pose = pose_trans(tuft_coords, p[0.7626, 0.8961, -0.0020, 0, 0, 0])
    movel(p[new_pose[0], new_pose[1], new_pose[2], current_pose[3], current_pose[4], current_pose[5]], a=1.2, v=0.0600)
    report_progress()
    set_digital_out(0, False)
    new_pose = pose_trans(tuft_coords, p[0.7626, 0.8961, 0.1500, 0, 0, 0])
    movel(p[new_pose[0], new_pose[1], new_pose[2], current_pose[3], current_pose[4], current_pose[5]], a=0.8, v=0.2000)
    report_progress()
    new_pose = pose_trans(tuft_coords, p[0.7646, 0.1539, 0.1500, 0, 0, 0])
    movel(p[new_pose[0], new_pose[1], new_pose[2], current_pose[3], current_pose[4], current_pose[5]], a=1.2, v=0.2000)
    report_progress()
    new_pose = pose_trans(tuft_coords, p[0.7646, 0.1539, -0.0020, 0, 0, 0])
    movel(p[new_pose[0], new_pose[1], new_pose[2], current_pose[3], current_pose[4], current_pose[5]], a=0.8, v=0.2000)
    report_progress()
    set_digital_out(0, True)
    new_pose = pose_trans(tuft_coords, p[0.7646, 0.8961, -0.0020, 0, 0, 0])
    movel(p[new_pose[0], new_pose[1], new_pose[2], current_pose[3], current_pose[4], current_pose[5]], a=1.2, v=0.0600)
    report_progress()
    set_digital_out(0, False)
    new_pose = pose_trans(tuft_coords, p[0.7646, 0.8961, 0.1500, 0, 0, 0])
    movel(p[new_pose[0], new_pose[1], new_pose[2], current_pose[3], current_pose[4], current_pose[5]], a=0.8, v=0.2000)
    report_progress()
    new_pose = pose_trans(tuft_coords, p[0.7665, 0.1539, 0.1500, 0, 0, 0])
    movel(p[new_pose[0], new_pose[1], new_pose[2], current_pose[3], current_pose[4], current_pose[5]], a=1.2, v=0.2000)
    report_progress()
    new_pose = pose_trans(tuft_coords, p[0.7665, 0.1539, -0.0020, 0, 0, 0])
    movel(p[new_pose[0], new_pose[1], new_pose[2], current_pose[3], current_pose[4], current_pose[5]], a=0.8, v=0.2000)
    report_progress()
    set_digital_out(0, True)
    new_pose = pose_trans(tuft_coords, p[0.7665, 0.8961, -0.0020, 0, 0, 0])
    movel(p[new_pose[0], new_pose[1], new_pose[2], current_pose[3], current_pose[4], current_pose[5]], a=1.2, v=0.0600)
    report_progress()
    set_digital_out(0, False)
    new_pose = pose_trans(tuft_coords, p[0.7665, 0.8961, 0.1500, 0, 0, 0])
    movel(p[new_pose[0], new_pose[1], new_pose[2], current_pose[3], current_pose[4], current_pose[5]], a=0.8, v=0.2000)
    report_progress()
    new_pose = pose_trans(tuft_coords, p[0.7685, 0.1539, 0.1500, 0, 0, 0])
    movel(p[new_pose[0], new_pose[1], new_pose[2], current_pose[3], current_pose[4], current_pose[5]], a=1.2, v=0.2000)
    report_progress()
    new_pose = pose_trans(tuft_coords, p[0.7685, 0.1539, -0.0020, 0, 0, 0])
    movel(p[new_pose[0], new_pose[1], new_pose[2], current_pose[3], current_pose[4], current_pose[5]], a=0.8, v=0.2000)
    report_progress()
    set_digital_out(0, True)
    new_pose = pose_trans(tuft_coords, p[0.7685, 0.8961, -0.0020, 0, 0, 0])
    movel(p[new_pose[0], new_pose[1], new_pose[2], current_pose[3], current_pose[4], current_pose[5]], a=1.2, v=0.0600)
    report_progress()
    set_digital_out(0, False)
    new_pose = pose_trans(tuft_coords, p[0.7685, 0.8961, 0.1500, 0, 0, 0])
    movel(p[new_pose[0], new_pose[1], new_pose[2], current_pose[3], current_pose[4], current_pose[5]], a=0.8, v=0.2000)
    report_progress()
    new_pose = pose_trans(tuft_coords, p[0.7704, 0.1559, 0.1500, 0, 0, 0])
    movel(p[new_pose[0], new_pose[1], new_pose[2], current_pose[3], current_pose[4], current_pose[5]], a=1.2, v=0.2000)
    report_progress()
    new_pose = pose_trans(tuft_coords, p[0.7704, 0.1559, -0.0020, 0, 0, 0])
    movel(p[new_pose[0], new_pose[1], new_pose[2], current_pose[3], current_pose[4], current_pose[5]], a=0.8, v=0.2000)
    report_progress()
    set_digital_out(0, True)
    new_pose = pose_trans(tuft_coords, p[0.7704, 0.8941, -0.0020, 0, 0, 0])
    movel(p[new_pose[0], new_pose[1], new_pose[2], current_pose[3], current_pose[4], current_pose[5]], a=1.2, v=0.0600)
    report_progress()
    set_digital_out(0, False)
    new_pose = pose_trans(tuft_coords, p[0.7704, 0.8941, 0.1500, 0, 0, 0])
    movel(p[new_pose[0], new_pose[1], new_pose[2], current_pose[3], current_pose[4], current_pose[5]], a=0.8, v=0.2000)
    report_progress()
    new_pose = pose_trans(tuft_coords, p[0.7724, 0.1559, 0.1500, 0, 0, 0])
    movel(p[new_pose[0], new_pose[1], new_pose[2], current_pose[3], current_pose[4], current_pose[5]], a=1.2, v=0.2000)
    report_progress()
    new_pose = pose_trans(tuft_coords, p[0.7724, 0.1559, -0.0020, 0, 0, 0])
    movel(p[new_pose[0], new_pose[1], new_pose[2], current_pose[3], current_pose[4], current_pose[5]], a=0.8, v=0.2000)
    report_progress()
    set_digital_out(0, True)
    new_pose = pose_trans(tuft_coords, p[0.7724, 0.8941, -0.0020, 0, 0, 0])
    movel(p[new_pose[0], new_pose[1], new_pose[2], current_pose[3], current_pose[4], current_pose[5]], a=1.2, v=0.0600)
    report_progress()
    set_digital_out(0, False)
    new_pose = pose_trans(tuft_coords, p[0.7724, 0.8941, 0.1500, 0, 0, 0])
    movel(p[new_pose[0], new_pose[1], new_pose[2], current_pose[3], current_pose[4], current_pose[5]], a=0.8, v=0.2000)
    report_progress()
    new_pose = pose_trans(tuft_coords, p[0.7743, 0.1559, 0.1500, 0, 0, 0])
    movel(p[new_pose[0], new_pose[1], new_pose[2], current_pose[3], current_pose[4], current_pose[5]], a=1.2, v=0.2000)
    report_progress()
    new_pose = pose_trans(tuft_coords, p[0.7743, 0.1559, -0.0020, 0, 0, 0])
    movel(p[new_pose[0], new_pose[1], new_pose[2], current_pose[3], current_pose[4], current_pose[5]], a=0.8, v=0.2000)
    report_progress()
    set_digital_out(0, True)
    new_pose = pose_trans(tuft_coords, p[0.7743, 0.8941, -0.0020, 0, 0, 0])
    movel(p[new_pose[0], new_pose[1], new_pose[2], current_pose[3], current_pose[4], current_pose[5]], a=1.2, v=0.0600)
    report_progress()
    set_digital_out(0, False)
    new_pose = pose_trans(tuft_coords, p[0.7743, 0.8941, 0.1500, 0, 0, 0])
    movel(p[new_pose[0], new_pose[1], new_pose[2], current_pose[3], current_pose[4], current_pose[5]], a=0.8, v=0.2000)
    report_progress()
    new_pose = pose_trans(tuft_coords, p[0.7762, 0.1559, 0.1500, 0, 0, 0])
    movel(p[new_pose[0], new_pose[1], new_pose[2], current_pose[3], current_pose[4], current_pose[5]], a=1.2, v=0.2000)
    report_progress()
    new_pose = pose_trans(tuft_coords, p[0.7762, 0.1559, -0.0020, 0, 0, 0])
    movel(p[new_pose[0], new_pose[1], new_pose[2], current_pose[3], current_pose[4], current_pose[5]], a=0.8, v=0.2000)
    report_progress()
    set_digital_out(0, True)
    new_pose = pose_trans(tuft_coords, p[0.7762, 0.8941, -0.0020, 0, 0, 0])
    movel(p[new_pose[0], new_pose[1], new_pose[2], current_pose[3], current_pose[4], current_pose[5]], a=1.2, v=0.0600)
    report_progress()
    set_digital_out(0, False)
    new_pose = pose_trans(tuft_coords, p[0.7762, 0.8941, 0.1500, 0, 0, 0])
    movel(p[new_pose[0], new_pose[1], new_pose[2], current_pose[3], current_pose[4], current_pose[5]], a=0.8, v=0.2000)
    report_progress()
    new_pose = pose_trans(tuft_coords, p[0.7782, 0.1559, 0.1500, 0, 0, 0])
    movel(p[new_pose[0], new_pose[1], new_pose[2], current_pose[3], current_pose[4], current_pose[5]], a=1.2, v=0.2000)
    report_progress()
    new_pose = pose_trans(tuft_coords, p[0.7782, 0.1559, -0.0020, 0, 0, 0])
    movel(p[new_pose[0], new_pose[1], new_pose[2], current_pose[3], current_pose[4], current_pose[5]], a=0.8, v=0.2000)
    report_progress()
    set_digital_out(0, True)
    new_pose = pose_trans(tuft_coords, p[0.7782, 0.8941, -0.0020, 0, 0, 0])
    movel(p[new_pose[0], new_pose[1], new_pose[2], current_pose[3], current_pose[4], current_pose[5]], a=1.2, v=0.0600)
    report_progress()
    set_digital_out(0, False)
    new_pose = pose_trans(tuft_coords, p[0.7782, 0.8941, 0.1500, 0, 0, 0])
    movel(p[new_pose[0], new_pose[1], new_pose[2], current_pose[3], current_pose[4], current_pose[5]], a=0.8, v=0.2000)
    report_progress()
    new_pose = pose_trans(tuft_coords, p[0.7801, 0.1559, 0.1500, 0, 0, 0])
    movel(p[new_pose[0], new_pose[1], new_pose[2], current_pose[3], current_pose[4], current_pose[5]], a=1.2, v=0.2000)
    report_progress()
    new_pose = pose_trans(tuft_coords, p[0.7801, 0.1559, -0.0020, 0, 0, 0])
    movel(p[new_pose[0], new_pose[1], new_pose[2], current_pose[3], current_pose[4], current_pose[5]], a=0.8, v=0.2000)
    report_progress()
    set_digital_out(0, True)
    new_pose = pose_trans(tuft_coords, p[0.7801, 0.8941, -0.0020, 0, 0, 0])
    movel(p[new_pose[0], new_pose[1], new_pose[2], current_pose[3], current_pose[4], current_pose[5]], a=1.2, v=0.0600)
    report_progress()
    set_digital_out(0, False)
    new_pose = pose_trans(tuft_coords, p[0.7801, 0.8941, 0.1500, 0, 0, 0])
    movel(p[new_pose[0], new_pose[1], new_pose[2], current_pose[3], current_pose[4], current_pose[5]], a=0.8, v=0.2000)
    report_progress()
    new_pose = pose_trans(tuft_coords, p[0.7821, 0.1559, 0.1500, 0, 0, 0])
    movel(p[new_pose[0], new_pose[1], new_pose[2], current_pose[3], current_pose[4], current_pose[5]], a=1.2, v=0.2000)
    report_progress()
    new_pose = pose_trans(tuft_coords, p[0.7821, 0.1559, -0.0020, 0, 0, 0])
    movel(p[new_pose[0], new_pose[1], new_pose[2], current_pose[3], current_pose[4], current_pose[5]], a=0.8, v=0.2000)
    report_progress()
    set_digital_out(0, True)
    new_pose = pose_trans(tuft_coords, p[0.7821, 0.8941, -0.0020, 0, 0, 0])
    movel(p[new_pose[0], new_pose[1], new_pose[2], current_pose[3], current_pose[4], current_pose[5]], a=1.2, v=0.0600)
    report_progress()
    set_digital_out(0, False)
    new_pose = pose_trans(tuft_coords, p[0.7821, 0.8941, 0.1500, 0, 0, 0])
    movel(p[new_pose[0], new_pose[1], new_pose[2], current_pose[3], current_pose[4], current_pose[5]], a=0.8, v=0.2000)
    report_progress()
    new_pose = pose_trans(tuft_coords, p[0.7840, 0.1559, 0.1500, 0, 0, 0])
    movel(p[new_pose[0], new_pose[1], new_pose[2], current_pose[3], current_pose[4], current_pose[5]], a=1.2, v=0.2000)
    report_progress()
    new_pose = pose_trans(tuft_coords, p[0.7840, 0.1559, -0.0020, 0, 0, 0])
    movel(p[new_pose[0], new_pose[1], new_pose[2], current_pose[3], current_pose[4], current_pose[5]], a=0.8, v=0.2000)
    report_progress()
    set_digital_out(0, True)
    new_pose = pose_trans(tuft_coords, p[0.7840, 0.8941, -0.0020, 0, 0, 0])
    movel(p[new_pose[0], new_pose[1], new_pose[2], current_pose[3], current_pose[4], current_pose[5]], a=1.2, v=0.0600)
    report_progress()
    set_digital_out(0, False)
    new_pose = pose_trans(tuft_coords, p[0.7840, 0.8941, 0.1500, 0, 0, 0])
    movel(p[new_pose[0], new_pose[1], new_pose[2], current_pose[3], current_pose[4], current_pose[5]], a=0.8, v=0.2000)
    report_progress()
    new_pose = pose_trans(tuft_coords, p[0.7860, 0.1559, 0.1500, 0, 0, 0])
    movel(p[new_pose[0], new_pose[1], new_pose[2], current_pose[3], current_pose[4], current_pose[5]], a=1.2, v=0.2000)
    report_progress()
    new_pose = pose_trans(tuft_coords, p[0.7860, 0.1559, -0.0020, 0, 0, 0])
    movel(p[new_pose[0], new_pose[1], new_pose[2], current_pose[3], current_pose[4], current_pose[5]], a=0.8, v=0.2000)
    report_progress()
    set_digital_out(0, True)
    new_pose = pose_trans(tuft_coords, p[0.7860, 0.8941, -0.0020, 0, 0, 0])
    movel(p[new_pose[0], new_pose[1], new_pose[2], current_pose[3], current_pose[4], current_pose[5]], a=1.2, v=0.0600)
    report_progress()
    set_digital_out(0, False)
    new_pose = pose_trans(tuft_coords, p[0.7860, 0.8941, 0.1500, 0, 0, 0])
    movel(p[new_pose[0], new_pose[1], new_pose[2], current_pose[3], current_pose[4], current_pose[5]], a=0.8, v=0.2000)
    report_progress()
    new_pose = pose_trans(tuft_coords, p[0.7879, 0.1559, 0.1500, 0, 0, 0])
    movel(p[new_pose[0], new_pose[1], new_pose[2], current_pose[3], current_pose[4], current_pose[5]], a=1.2, v=0.2000)
    report_progress()
    new_pose = pose_trans(tuft_coords, p[0.7879, 0.1559, -0.0020, 0, 0, 0])
    movel(p[new_pose[0], new_pose[1], new_pose[2], current_pose[3], current_pose[4], current_pose[5]], a=0.8, v=0.2000)
    report_progress()
    set_digital_out(0, True)
    new_pose = pose_trans(tuft_coords, p[0.7879, 0.8941, -0.0020, 0, 0, 0])
    movel(p[new_pose[0], new_pose[1], new_pose[2], current_pose[3], current_pose[4], current_pose[5]], a=1.2, v=0.0600)
    report_progress()
    set_digital_out(0, False)
    new_pose = pose_trans(tuft_coords, p[0.7879, 0.8941, 0.1500, 0, 0, 0])
    movel(p[new_pose[0], new_pose[1], new_pose[2], current_pose[3], current_pose[4], current_pose[5]], a=0.8, v=0.2000)
    report_progress()
    new_pose = pose_trans(tuft_coords, p[0.7899, 0.1559, 0.1500, 0, 0, 0])
    movel(p[new_pose[0], new_pose[1], new_pose[2], current_pose[3], current_pose[4], current_pose[5]], a=1.2, v=0.2000)
    report_progress()
    new_pose = pose_trans(tuft_coords, p[0.7899, 0.1559, -0.0020, 0, 0, 0])
    movel(p[new_pose[0], new_pose[1], new_pose[2], current_pose[3], current_pose[4], current_pose[5]], a=0.8, v=0.2000)
    report_progress()
    set_digital_out(0, True)
    new_pose = pose_trans(tuft_coords, p[0.7899, 0.8941, -0.0020, 0, 0, 0])
    movel(p[new_pose[0], new_pose[1], new_pose[2], current_pose[3], current_pose[4], current_pose[5]], a=1.2, v=0.0600)
    report_progress()
    set_digital_out(0, False)
    new_pose = pose_trans(tuft_coords, p[0.7899, 0.8941, 0.1500, 0, 0, 0])
    movel(p[new_pose[0], new_pose[1], new_pose[2], current_pose[3], current_pose[4], current_pose[5]], a=0.8, v=0.2000)
    report_progress()
    new_pose = pose_trans(tuft_coords, p[0.7918, 0.1559, 0.1500, 0, 0, 0])
    movel(p[new_pose[0], new_pose[1], new_pose[2], current_pose[3], current_pose[4], current_pose[5]], a=1.2, v=0.2000)
    report_progress()
    new_pose = pose_trans(tuft_coords, p[0.7918, 0.1559, -0.0020, 0, 0, 0])
    movel(p[new_pose[0], new_pose[1], new_pose[2], current_pose[3], current_pose[4], current_pose[5]], a=0.8, v=0.2000)
    report_progress()
    set_digital_out(0, True)
    new_pose = pose_trans(tuft_coords, p[0.7918, 0.8941, -0.0020, 0, 0, 0])
    movel(p[new_pose[0], new_pose[1], new_pose[2], current_pose[3], current_pose[4], current_pose[5]], a=1.2, v=0.0600)
    report_progress()
    set_digital_out(0, False)
    new_pose = pose_trans(tuft_coords, p[0.7918, 0.8941, 0.1500, 0, 0, 0])
    movel(p[new_pose[0], new_pose[1], new_pose[2], current_pose[3], current_pose[4], current_pose[5]], a=0.8, v=0.2000)
    report_progress()
    new_pose = pose_trans(tuft_coords, p[0.7937, 0.1579, 0.1500, 0, 0, 0])
    movel(p[new_pose[0], new_pose[1], new_pose[2], current_pose[3], current_pose[4], current_pose[5]], a=1.2, v=0.2000)
    report_progress()
    new_pose = pose_trans(tuft_coords, p[0.7937, 0.1579, -0.0020, 0, 0, 0])
    movel(p[new_pose[0], new_pose[1], new_pose[2], current_pose[3], current_pose[4], current_pose[5]], a=0.8, v=0.2000)
    report_progress()
    set_digital_out(0, True)
    new_pose = pose_trans(tuft_coords, p[0.7937, 0.8921, -0.0020, 0, 0, 0])
    movel(p[new_pose[0], new_pose[1], new_pose[2], current_pose[3], current_pose[4], current_pose[5]], a=1.2, v=0.0600)
    report_progress()
    set_digital_out(0, False)
    new_pose = pose_trans(tuft_coords, p[0.7937, 0.8921, 0.1500, 0, 0, 0])
    movel(p[new_pose[0], new_pose[1], new_pose[2], current_pose[3], current_pose[4], current_pose[5]], a=0.8, v=0.2000)
    report_progress()
    new_pose = pose_trans(tuft_coords, p[0.7957, 0.1579, 0.1500, 0, 0, 0])
    movel(p[new_pose[0], new_pose[1], new_pose[2], current_pose[3], current_pose[4], current_pose[5]], a=1.2, v=0.2000)
    report_progress()
    new_pose = pose_trans(tuft_coords, p[0.7957, 0.1579, -0.0020, 0, 0, 0])
    movel(p[new_pose[0], new_pose[1], new_pose[2], current_pose[3], current_pose[4], current_pose[5]], a=0.8, v=0.2000)
    report_progress()
    set_digital_out(0, True)
    new_pose = pose_trans(tuft_coords, p[0.7957, 0.8921, -0.0020, 0, 0, 0])
    movel(p[new_pose[0], new_pose[1], new_pose[2], current_pose[3], current_pose[4], current_pose[5]], a=1.2, v=0.0600)
    report_progress()
    set_digital_out(0, False)
    new_pose = pose_trans(tuft_coords, p[0.7957, 0.8921, 0.1500, 0, 0, 0])
    movel(p[new_pose[0], new_pose[1], new_pose[2], current_pose[3], current_pose[4], current_pose[5]], a=0.8, v=0.2000)
    report_progress()
    new_pose = pose_trans(tuft_coords, p[0.7976, 0.1579, 0.1500, 0, 0, 0])
    movel(p[new_pose[0], new_pose[1], new_pose[2], current_pose[3], current_pose[4], current_pose[5]], a=1.2, v=0.2000)
    report_progress()
    new_pose = pose_trans(tuft_coords, p[0.7976, 0.1579, -0.0020, 0, 0, 0])
    movel(p[new_pose[0], new_pose[1], new_pose[2], current_pose[3], current_pose[4], current_pose[5]], a=0.8, v=0.2000)
    report_progress()
    set_digital_out(0, True)
    new_pose = pose_trans(tuft_coords, p[0.7976, 0.8921, -0.0020, 0, 0, 0])
    movel(p[new_pose[0], new_pose[1], new_pose[2], current_pose[3], current_pose[4], current_pose[5]], a=1.2, v=0.0600)
    report_progress()
    set_digital_out(0, False)
    new_pose = pose_trans(tuft_coords, p[0.7976, 0.8921, 0.1500, 0, 0, 0])
    movel(p[new_pose[0], new_pose[1], new_pose[2], current_pose[3], current_pose[4], current_pose[5]], a=0.8, v=0.2000)
    report_progress()
    new_pose = pose_trans(tuft_coords, p[0.7996, 0.1579, 0.1500, 0, 0, 0])
    movel(p[new_pose[0], new_pose[1], new_pose[2], current_pose[3], current_pose[4], current_pose[5]], a=1.2, v=0.2000)
    report_progress()
    new_pose = pose_trans(tuft_coords, p[0.7996, 0.1579, -0.0020, 0, 0, 0])
    movel(p[new_pose[0], new_pose[1], new_pose[2], current_pose[3], current_pose[4], current_pose[5]], a=0.8, v=0.2000)
    report_progress()
    set_digital_out(0, True)
    new_pose = pose_trans(tuft_coords, p[0.7996, 0.8921, -0.0020, 0, 0, 0])
    movel(p[new_pose[0], new_pose[1], new_pose[2], current_pose[3], current_pose[4], current_pose[5]], a=1.2, v=0.0600)
    report_progress()
    set_digital_out(0, False)
    new_pose = pose_trans(tuft_coords, p[0.7996, 0.8921, 0.1500, 0, 0, 0])
    movel(p[new_pose[0], new_pose[1], new_pose[2], current_pose[3], current_pose[4], current_pose[5]], a=0.8, v=0.2000)
    report_progress()
    new_pose = pose_trans(tuft_coords, p[0.8015, 0.1579, 0.1500, 0, 0, 0])
